(* CoDeSys 2.3.9.47 project: myhome.pro *)
(* Libraries: TcDatabase.lib 17.3.10 13:31:12, COMlibV2.lib 24.2.14 12:45:46, TcSUPS.lib 4.12.14 19:04:14, TcBaseMath.lib 27.7.04 12:07:56, TcMath.lib 23.9.04 15:15:30, TcBABasic.lib 29.5.12 16:01:34, TcBase.lib 14.5.09 12:14:08, TcSystem.lib 24.2.16 14:35:18, TcUtilities.lib 3.2.16 16:08:58, TcEL6851.lib 22.4.12 13:04:27, STANDARD.LIB 5.6.98 12:03:02, TcpIp.lib 9.1.14 13:33:22 *)

(* Global variable list: Global_Variables *)
VAR_GLOBAL

	SYS_VKE_0:		BOOL	:=	FALSE;		(*SYSTEM ALWAYS 0*)
	SYS_VKE_1:		BOOL	:=	TRUE;		(*SYSTEM ALWAYS 1*)
	SYS_IBN_1:		BOOL	:=	TRUE;		(*SYSTEM IBN ALWAYS 1*)

	di_System_Time:	DINT;

	SYS_FPE_100MS:	BOOL	:=	FALSE;		(*SYSTEM TIME 0.1 sec*)
	SYS_FPE_200MS:	BOOL	:=	FALSE;		(*SYSTEM TIME 0.2 sec*)
	SYS_FPE_500MS:	BOOL	:=	FALSE;		(*SYSTEM TIME 0.5 sec*)
	SYS_FPE_1S:		BOOL	:=	FALSE;		(*SYSTEM TIME 1.0 sec*)
	SYS_FPE_2S:		BOOL	:=	FALSE;		(*SYSTEM TIME 2.0 sec*)

	SYS_TOG_100MS:	BOOL	:=	FALSE;		(*SYSTEM TIME 0.1 sec*)
	SYS_TOG_200MS:	BOOL	:=	FALSE;		(*SYSTEM TIME 0.2 sec*)
	SYS_TOG_500MS:	BOOL	:=	FALSE;		(*SYSTEM TIME 0.5 sec*)
	SYS_TOG_1S:		BOOL	:=	FALSE;		(*SYSTEM TIME 1.0 sec*)
	SYS_TOG_2S:		BOOL	:=	FALSE;		(*SYSTEM TIME 2.0 sec*)

	SYS_T_100MS:		TON;					(*SYSTEM TIME 0.1 sec*)
	SYS_T_200MS:		TON;					(*SYSTEM TIME 0.2 sec*)
	SYS_T_500MS:		TON;					(*SYSTEM TIME 0.5 sec*)
	SYS_T_1S:			TON;					(*SYSTEM TIME 1.0 sec*)
	SYS_T_2S:			TON;					(*SYSTEM TIME 2.0 sec*)

	AX_FPE_100MS:	R_TRIG;				(*SYSTEM AUX FPE 0.1 sec*)
	AX_FPE_200MS:	R_TRIG;				(*SYSTEM AUX FPE 0.2 sec*)
	AX_FPE_500MS:	R_TRIG;				(*SYSTEM AUX FPE 0.5 sec*)
	AX_FPE_1S:		R_TRIG;				(*SYSTEM AUX FPE 1.0 sec*)
	AX_FPE_2S:		R_TRIG;				(*SYSTEM AUX FPE 2.0 sec*)

	bNightMode:	BOOL := FALSE;	(*limits Brightness if active*)
	fbTime : FB_LocalSystemTime := ( bEnable := TRUE, dwCycle := 1 );

(*DIGITAL INPUTS/Outputs*)
	(*SPS Switch 01 Arbeitsraum*)
	DI_S01_1 	AT %IX50.0 : BOOL;	(*Function Left 1*)
	DI_S01_2	AT %IX50.1 : BOOL;	(*Function Right 1*)
	DI_S01_3	AT %IX50.2 : BOOL;	(*Function Left 2*)
	DI_S01_4	AT %IX50.3 : BOOL;	(*Function Right 2*)
	DI_S01_5	AT %IX50.4 : BOOL;	(*Function Left 3*)
	DI_S01_6	AT %IX50.5 : BOOL;	(*Function Right 3*)
	DO_S01_0 	AT %QX50.0 : BOOL;	(*Status LED Left 1*)
	DO_S01_1 	AT %QX50.1 : BOOL;	(*Status LED Right 1*)
	DO_S01_2 	AT %QX50.2 : BOOL;	(*Status LED Left 2*)
	DO_S01_3 	AT %QX50.3 : BOOL;	(*Status LED Right 2*)
	DO_S01_4 	AT %QX50.4 : BOOL;	(*Status LED Left 3*)
	DO_S01_5 	AT %QX50.5 : BOOL;	(*Status LED Right 3*)
	DO_S01_6 	AT %QX50.6 : BOOL;	(*Background LED*)

	(*SPS Switch 02 Wohnzimmer*)
	DI_S02_1 	AT %IX50.6 : BOOL;	(*Function Left 1*)
	DI_S02_2	AT %IX50.7 : BOOL;	(*Function Right 1*)
	DI_S02_3	AT %IX51.0 : BOOL;	(*Function Left 2*)
	DI_S02_4	AT %IX51.1 : BOOL;	(*Function Right 2*)
	DI_S02_5	AT %IX51.2 : BOOL;	(*Function Left 3*)
	DI_S02_6	AT %IX51.3 : BOOL;	(*Function Right 3*)
	DO_S02_0 	AT %QX50.7 : BOOL;	(*Status LED Left 1*)
	DO_S02_1 	AT %QX51.0 : BOOL;	(*Status LED Right 1*)
	DO_S02_2 	AT %QX51.1 : BOOL;	(*Status LED Left 2*)
	DO_S02_3 	AT %QX51.2 : BOOL;	(*Status LED Right 2*)
	DO_S02_4 	AT %QX51.3 : BOOL;	(*Status LED Left 3*)
	DO_S02_5 	AT %QX51.4 : BOOL;	(*Status LED Right 3*)
	DO_S02_6 	AT %QX51.5 : BOOL;	(*Background LED*)

	(*DOUBLE Switch 03*)
	DI_S03_1 	AT %IX51.4 : BOOL;	(*Function Left*)
	DI_S03_2 	AT %IX51.5 : BOOL;	(*Function Right*)

	(*DOUBLE Switch 04*)
	DI_S04_1 	AT %IX51.6 : BOOL;	(*Function Left*)
	DI_S04_2 	AT %IX51.7 : BOOL;	(*Function Right*)

	(*SPS Switch 05 Schlafzimmer Bett Links*)
	DI_S05_1 	AT %IX52.0 : BOOL;	(*Function Left 1*)
	DI_S05_2	AT %IX52.1 : BOOL;	(*Function Right 1*)
	DI_S05_3	AT %IX52.2 : BOOL;	(*Function Left 2*)
	DI_S05_4	AT %IX52.3 : BOOL;	(*Function Right 2*)
	DI_S05_5	AT %IX52.4 : BOOL;	(*Function Left 3*)
	DI_S05_6	AT %IX52.5 : BOOL;	(*Function Right 3*)
	DO_S05_0 	AT %QX51.6 : BOOL;	(*Status LED Left 1*)
	DO_S05_1 	AT %QX51.7 : BOOL;	(*Status LED Right 1*)
	DO_S05_2 	AT %QX52.0 : BOOL;	(*Status LED Left 2*)
	DO_S05_3 	AT %QX52.1 : BOOL;	(*Status LED Right 2*)
	DO_S05_4 	AT %QX52.2 : BOOL;	(*Status LED Left 3*)
	DO_S05_5 	AT %QX52.3 : BOOL;	(*Status LED Right 3*)
	DO_S05_6 	AT %QX52.4 : BOOL;	(*Background LED*)

	(*SPS Switch 06 Schlafzimmer Bett Rechts*)
	DI_S06_1 	AT %IX52.6 : BOOL;	(*Function Left 1*)
	DI_S06_2	AT %IX52.7 : BOOL;	(*Function Right 1*)
	DI_S06_3	AT %IX53.0 : BOOL;	(*Function Left 2*)
	DI_S06_4	AT %IX53.1 : BOOL;	(*Function Right 2*)
	DI_S06_5	AT %IX53.2 : BOOL;	(*Function Left 3*)
	DI_S06_6	AT %IX53.3 : BOOL;	(*Function Right 3*)
	DO_S06_0 	AT %QX52.5 : BOOL;	(*Status LED Left 1*)
	DO_S06_1 	AT %QX52.6 : BOOL;	(*Status LED Right 1*)
	DO_S06_2 	AT %QX52.7 : BOOL;	(*Status LED Left 2*)
	DO_S06_3 	AT %QX53.0 : BOOL;	(*Status LED Right 2*)
	DO_S06_4 	AT %QX53.1 : BOOL;	(*Status LED Left 3*)
	DO_S06_5 	AT %QX53.2 : BOOL;	(*Status LED Right 3*)
	DO_S06_6 	AT %QX53.3 : BOOL;	(*Background LED*)

	(*DOUBLE Switch 07*)
	DI_S07_1 	AT %IX53.4 : BOOL;	(*Function Left*)
	DI_S07_2 	AT %IX53.5 : BOOL;	(*Function Right*)

	(*SINGLE Switch 08*)
	DI_S08	 	AT %IX53.6 : BOOL;	(*Function*)

	(*SINGLE Switch 09*)
	DI_S09	 	AT %IX53.7 : BOOL;	(*Function*)

	(*SINGLE Switch 10*)
	DI_S10	 	AT %IX54.0 : BOOL;	(*Function*)

	(*SINGLE Swith 11*)
	DI_S11	 	AT %IX54.1 : BOOL;	(*Function*)

	(*MOTION Swith 01*)
	DI_BM1	 	AT %IX54.3 : BOOL;	(*Function*)

	(*MOTION Swith 02*)
	DI_BM2	 	AT %IX54.4 : BOOL;	(*Function*)

	(*MOTION Swith 03*)
	DI_BM3	 	AT %IX54.5 : BOOL;	(*Function*)

	(*Relais*)
	DO_NN_K01	AT %QX54.0 : BOOL;	(*Relais Netzteil Arbeitsraum*)
	DO_NN_K02	AT %QX54.1 : BOOL;	(*Relais Steckdosen Arbeitsraum*)
	DO_NN_K03	AT %QX54.2 : BOOL;	(*Relais Netzteil Wohnzimmer*)
	DO_NN_K04	AT %QX54.3 : BOOL;	(*Relais Steckdosen Fernseher*)
	DO_NN_K05	AT %QX54.4 : BOOL;	(*Relais Netzteil Küche*)
	DO_NN_K06	AT %QX54.5 : BOOL;	(*Relais Netzteil Zimmer / Schlafzimmer*)
	DO_NN_K07	AT %QX54.6 : BOOL;	(*Relais Netzteil WC, Gang und Abstellraum*)
	DO_NN_K08	AT %QX54.7 : BOOL;	(*Relais Licht Bad*)
	DO_NN_K09	AT %QX53.6 : BOOL;	(*Relais Ventilator WC*)
	DO_NN_K10	AT %QX53.7 : BOOL;	(*Relais Reserve*)

	DO_NAS_BACKUP_ON_OFF	AT %QX53.4 : BOOL;	(*Relais NAS-Backup Pulse Power Switch*)
	DO_NAS_ON_OFF	AT %QX53.5 : BOOL;	(*Relais  NAS Pulse Power Switch*)

	fbPowerPC:PRG_FB_PULSE_SWITCH;
	fbPowerNAS:PRG_FB_PULSE_SWITCH;
	fbPowerNASBackup:PRG_FB_PULSE_SWITCH;

(* DMX Line *)
	fbEL6851Communication	:	FB_EL6851Communication;
	stDMXInDataLinie01               AT %I*	:	ST_EL6851InData;
	stDMXOutDataLinie01              AT %Q*	:	ST_EL6851OutData;
	stCommandBuffer01						:	ST_DMXCommandBuffer;
	arrDMXProcessData						:	ARRAY [1..512] OF BYTE;

(* 	I/O variables for a KL6001 terminal*)
	COMin_KL6001			AT %I* 	: KL6inData22B;		(* linked to the KL6001 in the TwinCAT System Manager *)
	COMout_KL6001		AT %Q*	: KL6outData22B;	(* linked to the KL6001 in the TwinCAT System Manager *)
	RxBuffer2: ComBuffer;	(* Receive data buffer; used with all receive function blocks *)
	TxBuffer2: ComBuffer;	(* Transmit data buffer; used with all receive function blocks *)

	COMin_COM4			AT %I* 	: KL6inData22B;		(* linked to the KL6001 in the TwinCAT System Manager *)
	COMout_COM4		AT %Q*	: KL6outData22B;	(* linked to the KL6001 in the TwinCAT System Manager *)

(*	FIFO for Trend if Database is off - Max 1 Week can be saved with 1 value every Minute*)
	TemperatureSchlafzimmerFIFO: PRG_FIFO_10080;
	TemperatureKinderzimmerFIFO: PRG_FIFO_10080;
	TemperatureKuecheFIFO: PRG_FIFO_10080;
	HumiditySchlafzimmerFIFO: PRG_FIFO_10080;
	HumidityKinderzimmerFIFO: PRG_FIFO_10080;
	HumidityKuecheFIFO: PRG_FIFO_10080;

	TemperatureTerrariumLinksFIFO: PRG_FIFO_10080;
	HumidityTerrariumLinksFIFO: PRG_FIFO_10080;
	TemperatureTerrariumRechtsFIFO: PRG_FIFO_10080;
	HumidityTerrariumRechtsFIFO: PRG_FIFO_10080;

(* TEST UDP*)
	g_sTcIpConnSvrAddr								:  T_AmsNetId := '10.0.0.6';

	(* Some project specific error codes *)
	PLCPRJ_ERROR_SENDFIFO_OVERFLOW		: UDINT := 16#8103;
	PLCPRJ_ERROR_RECFIFO_OVERFLOW		: UDINT := 16#8104;

END_VAR

VAR_GLOBAL CONSTANT
	bLogDebugMessages								: BOOL := TRUE;

	MAX_CLIENT_CONNECTIONS						: UDINT(1..20) := 5;
	MAX_PLCPRJ_RXBUFFER_SIZE					: UDINT := 1000;


	PLCPRJ_RECONNECT_TIME						: TIME := T#3s;
	PLCPRJ_SEND_CYCLE_TIME						: TIME := T#1s;
	PLCPRJ_ACCEPT_POLLING_TIME					: TIME := T#1s;

	PLCPRJ_RECEIVE_POLLING_TIME		 			: TIME := T#1s;
	PLCPRJ_RECEIVE_TIMEOUT						: TIME := T#50s;

	(* Some project specific error codes *)
	PLCPRJ_ERROR_RECEIVE_BUFFER_OVERFLOW	: UDINT := 16#8101; (* receive buffer overflow*)
	PLCPRJ_ERROR_RECEIVE_TIMEOUT				: UDINT := 16#8102;(* receive timeout error *)

END_VAR

(* Global variable list: TwinCAT_Configuration *)
(* Generated automatically by TwinCAT - (read only) *)
VAR_CONFIG
	.stDMXInDataLinie01 AT %IB56 : ST_EL6851InData;
	.stDMXOutDataLinie01 AT %QB56 : ST_EL6851OutData;
	.COMin_KL6001 AT %IB132 : KL6inData22B;
	.COMout_KL6001 AT %QB576 : KL6outData22B;
END_VAR

(* Data type *)
TYPE E_ClientServerSteps :
(
	UDP_STATE_IDLE		:= 0,
	UDP_STATE_CREATE_START,
	UDP_STATE_CREATE_WAIT,
	UDP_STATE_SEND_START,
	UDP_STATE_SEND_WAIT,
	UDP_STATE_RECEIVE_START,
	UDP_STATE_RECEIVE_WAIT,
	UDP_STATE_CLOSE_START,
	UDP_STATE_CLOSE_WAIT,
	UDP_STATE_ERROR
);
END_TYPE

(* Data type *)
TYPE E_ClientSteps :
(
	CLIENT_STATE_IDLE,
	CLIENT_STATE_CONNECT_START,
	CLIENT_STATE_CONNECT_WAIT,
	CLIENT_STATE_DATAEXCHA_START,
	CLIENT_STATE_DATAEXCHA_WAIT,
	CLIENT_STATE_CLOSE_START,
	CLIENT_STATE_CLOSE_WAIT,
	CLIENT_STATE_ERROR
);
END_TYPE

(* Data type *)
TYPE E_DataExchaSteps :
(
	DATAEXCHA_STATE_IDLE,
	DATAEXCHA_STATE_SEND_START,
	DATAEXCHA_STATE_SEND_WAIT,
	DATAEXCHA_STATE_RECEIVE_START,
	DATAEXCHA_STATE_RECEIVE_WAIT,
	DATAEXCHA_STATE_ERROR
);
END_TYPE

(* Data type *)
TYPE E_SampleState :(
        eIdle := 0,
        eWriteAppend := 1,
        eWriteUpdate := 2,
        eWriteRingBuffer := 3
);
END_TYPE

(* Data type *)
TYPE E_ServerSteps :
(
	SERVER_STATE_IDLE,
	SERVER_STATE_LISTENER_OPEN_START,
	SERVER_STATE_LISTENER_OPEN_WAIT,
	SERVER_STATE_REMOTE_CLIENTS_COMM,
	SERVER_STATE_REMOTE_CLIENTS_CLOSE,
	SERVER_STATE_LISTENER_CLOSE_START,
	SERVER_STATE_LISTENER_CLOSE_WAIT,
	SERVER_STATE_ERROR
);
END_TYPE

(* Data type *)
TYPE E_SQLStatement :(
        eSQL_INSERT := 0,
        eSQL_SELECT := 1
);
END_TYPE

(* Data type *)
TYPE ST_FifoEntry :
STRUCT
	sRemoteHost		: STRING(15);		(* Remote address. String containing an (Ipv4) Internet Protocol dotted address. *)
	nRemotePort		: UDINT;			(* Remote Internet Protocol (IP) port. *)
	msg				: STRING;			(* Udp packet data *)
END_STRUCT
END_TYPE

(* Data type *)
TYPE ST_Record :
STRUCT
        Timestamp : DT;
        PLC_Value1 : REAL;
        PLC_Value2 : REAL;
        PLC_Value3 : REAL;
        PLC_Value4 : STRING;
END_STRUCT
END_TYPE

(* Data type *)
TYPE T_TimeStampLength : STRING(19);
END_TYPE

(* Data type *)
TYPE Type_HSV :
STRUCT
	Hue	:			REAL;
	Saturation:		REAL:= 100.0;
	Brightness:		REAL:=100.0;
END_STRUCT
END_TYPE

(* Data type *)
TYPE Type_LED :
STRUCT
	Switch_ON:			BOOL;
	Switch_RANDOM:		BOOL;
	bLight:				BOOL;
	Config:				Type_LED_CONFIG;
	Value:				REAL:=100;
	Brightness:			BYTE;
	fbDimmer2Switch: FB_Dimmer2Switch;
	fpSwitchOnOff: F_TRIG;
END_STRUCT
END_TYPE

(* Data type *)
TYPE Type_LED_CONFIG :
STRUCT
	tDimmTime: 		REAL	:= 5000;
	bDimmOnMode:	BOOL	:= TRUE;
	tDimmOnTime:		REAL	:= 500;
	bDimmOffMode:	BOOL	:= TRUE;
	tDimmOffTime:		REAL	:= 1000;
	Brightness_MAX	:REAL:=255;
END_STRUCT
END_TYPE

(* Data type *)
TYPE Type_LED_RGB :
STRUCT
	Hue				:REAL;
	Saturation			:REAL:= 100.0;
	Brightness			:REAL:=100;
	Switch_ON			:BOOL;
	Switch_RANDOM	:BOOL;
	bLight:			BOOL;
	Config				:Type_LED_RGB_CONFIG;
	Red					:BYTE;
	Green				:BYTE;
	Blue					:BYTE;
END_STRUCT
END_TYPE

(* Data type *)
TYPE Type_LED_RGB_CONFIG :
STRUCT
	Speed_RANDOM	:REAL;

	tDimmTime: 		REAL	:= 5000;
	bDimmOnMode:	BOOL	:= TRUE;
	tDimmOnTime:		REAL	:= 500;
	bDimmOffMode:	BOOL	:= TRUE;
	tDimmOffTime:		REAL	:= 1000;
END_STRUCT
END_TYPE

(* Data type *)
TYPE Type_LED_RGB_with_FB :
STRUCT
	Hue				:REAL;
	Saturation			:REAL:= 100.0;
	Brightness			:REAL:=100;
	Switch_ON			:BOOL;
	Switch_RANDOM	:BOOL;
	bLight:			BOOL;
	Config				:Type_LED_RGB_CONFIG;
	Red					:BYTE;
	Green				:BYTE;
	Blue					:BYTE;
	fbDimmer2Switch: FB_Dimmer2Switch;
	fpSwitchOnOff: F_TRIG;
END_STRUCT
END_TYPE

(* Data type *)
TYPE Type_SCENE_CONFIG :
STRUCT
	tDimmTime: 		REAL	:= 5000;
	bDimmOnMode:	BOOL	:= TRUE;
	tDimmOnTime:		REAL	:= 500;
	bDimmOffMode:	BOOL	:= TRUE;
	tDimmOffTime:		REAL	:= 1000;
END_STRUCT
END_TYPE

(* Data type *)
TYPE Type_SCENE_WZ :
STRUCT
	tyMirror1 : Type_LED_RGB;
	tyMirror2 : Type_LED_RGB;
	tyMirror3 : Type_LED_RGB;
(*tyCeiling : Type_LED_RGB;*)
END_STRUCT
END_TYPE

(* POU MAIN, ST *)
PROGRAM MAIN
VAR
	nCount 						: UDINT;
	tGlobOff:	TON;
	tGlobOffLong:	TOF;
	fnGlobOff: R_TRIG;

	nBrightness1:BYTE;
	nBrightness2:BYTE;
	nBrightness3:BYTE;
	nBrightness4:BYTE;
	nBrightness5:BYTE;
	nBrightness6:BYTE;
	nBrightness7:BYTE;
	nBrightness8:BYTE;
	nBrightness9:BYTE;

	READ_TEMP_HUM:SYS_03_READ_TEMP_HUM;
	COMM_XMC : SYS_02_COMM_XMC;

END_VAR
SYS_00_BASICS();
READ_TEMP_HUM(bEnable:=TRUE );
COMM_XMC(bEnable:=TRUE );

tGlobOff(IN:= DI_S05_6 OR DI_S06_6, PT:= T#2s);
fnGlobOff(CLK:= tGlobOff.Q );
tGlobOffLong(IN:= fnGlobOff.Q, PT:= T#4s);

(*Aufruf Wohnräume*)
ROOM_01_ARBEITSZIMMER(ibGlobOff:= fnGlobOff.Q, ibGlobOffLong:= tGlobOffLong.Q);
ROOM_02_WOHNZIMMER(ibGlobOff:= fnGlobOff.Q, ibGlobOffLong:= tGlobOffLong.Q, irTemperature:=READ_TEMP_HUM.Temp[1], irHumidity:=READ_TEMP_HUM.Humidity[1]);
ROOM_03_KUECHE(ibGlobOff:= fnGlobOff.Q, ibGlobOffLong:= tGlobOffLong.Q, irTemperature:=READ_TEMP_HUM.Temp[4], irHumidity:=READ_TEMP_HUM.Humidity[4]);
ROOM_04_ZIMMER(ibGlobOff:= fnGlobOff.Q, ibGlobOffLong:= tGlobOffLong.Q, irTemperature:=READ_TEMP_HUM.Temp[1], irHumidity:=READ_TEMP_HUM.Humidity[1], irTemperatureSZ:=READ_TEMP_HUM.Temp[5], irHumiditySZ:=READ_TEMP_HUM.Humidity[5]);
ROOM_05_WC_GANG(ibGlobOff:= fnGlobOff.Q, ibGlobOffLong:= tGlobOffLong.Q);

DO_S05_5:=	(ROOM_01_ARBEITSZIMMER.obDevOn OR ROOM_02_WOHNZIMMER.obDevOn OR
			ROOM_03_KUECHE.obDevOn OR ROOM_04_ZIMMER.obDevOn OR
			ROOM_05_WC_GANG.obDevOn) AND (fbTime.systemTime.wHour < 6 OR fbTime.systemTime.wHour >= 22);

DO_S06_5:=	(ROOM_01_ARBEITSZIMMER.obDevOn OR ROOM_02_WOHNZIMMER.obDevOn OR
			ROOM_03_KUECHE.obDevOn OR ROOM_04_ZIMMER.obDevOn OR
			ROOM_05_WC_GANG.obDevOn) AND (fbTime.systemTime.wHour < 6 OR fbTime.systemTime.wHour >= 22);

arrDMXProcessData[128] := nBrightness1;
arrDMXProcessData[129] := nBrightness2;
arrDMXProcessData[130] := nBrightness3;
arrDMXProcessData[131] := nBrightness4;
arrDMXProcessData[132] := nBrightness5;
arrDMXProcessData[133] := nBrightness6;
arrDMXProcessData[134] := nBrightness7;
arrDMXProcessData[135] := nBrightness8;

fbEL6851Communication(	wSourceManufacturerID := 16#42_41,
						dwSourceDeviceID := 16#12_13_14_15,
						bEnableSendingData := TRUE,
						bSetCycleMode := TRUE,
						bSendDefaultData := FALSE,
						uiDataLength := 512,
						dwOptions := 0,
						stEL6851InData := stDMXInDataLinie01,
						stEL6851OutData := stDMXOutDataLinie01,
						stCommandBuffer := stCommandBuffer01,
						arrProcessData := arrDMXProcessData);

fbTime();

SYS_01_TREND(
	irTemperatureSchlafzimmer:= READ_TEMP_HUM.Temp[5],
	irHumiditySchlafzimmer:= READ_TEMP_HUM.Humidity[5],
	irTemperatureKinderzimmer:= READ_TEMP_HUM.Temp[1],
	irHumidityKinderzimmer:= READ_TEMP_HUM.Humidity[1],
	irTemperatureKueche:= READ_TEMP_HUM.Temp[4],
	irHumidityKueche:= READ_TEMP_HUM.Humidity[4],
	irTemperatureTerrariumLinks:=COMM_XMC.TemperatureTerrariumLinks,
	irHumidityTerrariumLinks:=COMM_XMC.HumidityTerrariumLinks,
	irTemperatureTerrariumRechts:=COMM_XMC.TemperatureTerrariumRechts,
	irHumidityTerrariumRechts:=COMM_XMC.HumidityTerrariumRechts);
END_PROGRAM

(* POU General/SYS_03_READ_TEMP_HUM, ST *)
FUNCTION_BLOCK SYS_03_READ_TEMP_HUM
VAR_INPUT
	bEnable:BOOL;
END_VAR
VAR_OUTPUT
END_VAR
VAR
	Timer: TON;
	iActSensorNumber:UINT:=1;
	iNumberOfSensors:UINT:=5;
	RequestString:STRING;
	Send: SendString;
	SendBusy: BOOL;
	SendErrorID: ComError_t;

	Receive: ReceiveString;
	ReceivedString: STRING;
	LastReceivedString: STRING;
	StringReceived: BOOL;
	ReceiveBusy: BOOL;
	ReceiveError: BOOL;
	ReceiveErrorID: ComError_t;
	ReceiveTimeout: BOOL;
	ReceiveCounter: UDINT;
END_VAR
VAR PERSISTENT
	TempOffset: ARRAY [1..10] OF REAL := 0;
	Temp: ARRAY [1..10] OF REAL := 0;
	RecTempStr: ARRAY [1..10] OF STRING;
	Humidity: ARRAY [1..10] OF REAL := 0;
	RecHumidityStr: ARRAY [1..10] OF STRING;
END_VAR
(*==================================================================
	Call the send block every second to repeat the transmission.
	Also call the block as long as it is busy to finish a transmission.
*)

TempOffset[1]:=-1.2;
TempOffset[2]:=-2.6;
TempOffset[3]:=-1.6;
TempOffset[4]:=-2.6;
TempOffset[5]:=-1;

Timer(IN:=bEnable, PT:=T#1s);

IF Timer.Q OR Send.Busy THEN

	iActSensorNumber:=iActSensorNumber+1;
	IF iActSensorNumber > iNumberOfSensors THEN
		iActSensorNumber:=1;
	END_IF

	RequestString:= CONCAT('s',UINT_TO_STRING(iActSensorNumber));

	Send(	SendString:= RequestString,
			TXbuffer:= TxBuffer2,	(* see global variables *)
			Busy=> SendBusy,
			Error=> SendErrorID);

	Timer(IN:=FALSE); (* reset timer *)
END_IF

(*==================================================================
	Receive string data 
	The block receives any data strings beginning with a STX ($02) character and 
	ending with an ETX ($03) character.	
*)
Receive(
	Prefix:= '$02',
	Suffix:= '$03',
	Timeout:= T#1s,
	ReceivedString:= ReceivedString,
	RXbuffer:= RxBuffer2,
	StringReceived=> StringReceived,
	Busy=> ReceiveBusy,
	Error=> ReceiveErrorID,
	RxTimeout=> ReceiveTimeout );
IF StringReceived THEN
	ReceiveCounter := ReceiveCounter + 1;
	LastReceivedString := ReceivedString;

	(*Extract Temperatur Value from received String*)
	(*Nr. 4 = Küche, Nr.5 = Schlafzimmer*)
	RecTempStr[iActSensorNumber] := MID (ReceivedString,4,5);
	Temp[iActSensorNumber]:=STRING_TO_REAL(RecTempStr[iActSensorNumber] )+TempOffset[iActSensorNumber];

	(*Extract Humidity Value from received String*)
	RecHumidityStr[iActSensorNumber] := MID (ReceivedString,4,16);
	Humidity[iActSensorNumber]:=STRING_TO_REAL(RecHumidityStr[iActSensorNumber] );
END_IF


(*==================================================================
	Background communication with the KL6001 terminal.
	Please check the FAST program where the background communication with the
	KL6001 terminal is processed in a separate fast task. A fast task is in this case 
	necessary to guarantee an acceptable transfer rate.
*)
END_FUNCTION_BLOCK

(* POU General/SYS_02_COMM_XMC, ST *)
FUNCTION_BLOCK SYS_02_COMM_XMC
VAR_INPUT
	bEnable:BOOL;
END_VAR
VAR_OUTPUT
END_VAR
VAR
	Timer: TON;
	fpSend: R_TRIG;
	fpSwitchRollo: R_TRIG;
	fpAutoUp: R_TRIG;
	CommandString:STRING;
	Send: SendString;
	SendBusy: BOOL;
	SendErrorID: ComError_t;

	Receive: ReceiveString;
	ReceivedString: STRING;
	LastReceivedString: STRING;
	StringReceived: BOOL;
	ReceiveBusy: BOOL;
	ReceiveError: BOOL;
	ReceiveErrorID: ComError_t;
	ReceiveTimeout: BOOL;
	ReceiveCounter: UDINT;

	(* communication buffer between application and SerialLineControl *)
	RxBuffer		:ComBuffer;
	TxBuffer		:ComBuffer;

	(* serial line control *)
	fbLineCtrlAds	:SerialLineControlADS;
	bAdsError		:BOOL;
	nAdsErrorID		:UDINT;
	sNetId			:T_AmsNetId;
	stSerialCfg		:ComSerialConfig;

	bSendCommand:BOOL;

	boolRolloUp: BOOL := TRUE;
	boolRolloDown: BOOL;
	boolRolloCoUp: BOOL;
	boolRolloCoDown: BOOL;
	TON_DriveTime : TON;

	nRolloStat:INT:=10;
	nFindString : INT;


	TemperatureTerrariumLinks: REAL;
	HumidityTerrariumLinks: REAL;
	TemperatureTerrariumRechts: REAL;
	HumidityTerrariumRechts: REAL;
	tmpString: STRING;
	tmpString1: STRING;
END_VAR
VAR CONSTANT
	bRolloAutoControl:BOOL;
	nRolloAutoOpenTime:INT;
	ROLLO_UP : INT :=10;
	ROLLO_DRIVE_UP : INT := 11;
	ROLLO_DOWN : INT := 20;
	ROLLO_DRIVE_DOWN: INT := 21;
END_VAR
stSerialCfg.ComPort := 4;

fbLineCtrlAds(
	Connect:= bEnable,
	SerialCfg:= stSerialCfg,
	NetId:= sNetId,
	Timeout:= ,
	TxBuffer:= TxBuffer,
	RxBuffer:= RxBuffer,
	PortOpened=> ,
	Error=> bAdsError,
	ErrorID=> nAdsErrorID,
	Busy=> ,
	TxBufCount=> ,
	RxBufCount=> );

(*==================================================================
	Senden der Befehle	
	Befehle: CO_U: Rollo hoch, CU_D: Rollo runter, CO_S: Rollo Stop
*)
fpSend(CLK:=bSendCommand);
IF fpSend.Q OR Send.Busy OR Timer.Q THEN
	Send(	SendString:= CommandString,
			TXbuffer:= TxBuffer,	(* see global variables *)
	Busy=> SendBusy,
	Error=> SendErrorID);

	Timer(IN:=FALSE, PT:=T#10s);
END_IF

(*==================================================================
	Steuerung der Rollo
	Rauf-, Runterfahren und Stop	
*)

(*Schalter Rollo*)
fpSwitchRollo(CLK:= DI_S02_6);
Timer(IN:=bSendCommand, PT:=T#10s);

IF StringReceived THEN
	ReceiveCounter := ReceiveCounter + 1;
	LastReceivedString := ReceivedString;
END_IF

(*Um 10 Uhr automatisch die Rollo öffnen*)
fpAutoUp(CLK:= (fbTime.systemTime.wHour = nRolloAutoOpenTime) AND bRolloAutoControl);
IF fpAutoUp.Q THEN
	nRolloStat := ROLLO_DOWN;
END_IF


CASE nRolloStat OF
	ROLLO_UP:
		(*Rollo ist oben, starte Runterfahren bei Knopfdruck*)
		IF fpSwitchRollo.Q THEN
			CommandString:= 'CO_D';
			bSendCommand := TRUE;
		END_IF

		(*Befehl ist gesendet, warte auf Rückmeldung*)
		IF StringReceived THEN
			nFindString := FIND(LastReceivedString, 'CO_D');
			IF nFindString > 0 THEN
				nRolloStat := ROLLO_DRIVE_DOWN;
			END_IF
			bSendCommand := FALSE;
		END_IF

	ROLLO_DRIVE_DOWN:
		(*Starte Zeit*)
		IF NOT bSendCommand THEN
			TON_DriveTime(IN:= TRUE, PT:=T#21s);
		END_IF
		DO_S02_5 := SYS_TOG_200MS;

		(*Wenn während dem Fahren der Knopf gedrückt wird, dann wird Stop gesendet.*)
		IF fpSwitchRollo.Q THEN
			CommandString:= 'CO_S';
			bSendCommand := TRUE;
		END_IF

		(*Zeit abgelaufen, Rollo ist oben*)
		IF TON_DriveTime.Q THEN
			TON_DriveTime(IN:= FALSE);
			nRolloStat := ROLLO_DOWN;
			DO_S02_5:=FALSE;
		END_IF

		(*Wenn Stop Befehl gesendet wurde, dann springe zu status ROLLO_UP, dass beim nächsten druck das Rollo weiter nach unten fährt*)
		IF StringReceived THEN
			nFindString := FIND(LastReceivedString, 'CO_S');
			IF nFindString > 0 THEN
				nRolloStat := ROLLO_UP;
				DO_S02_5:=FALSE;
			END_IF
			bSendCommand := FALSE;
		END_IF

	ROLLO_DOWN:
		(*Rollo ist unten, starte Raufahren bei Knopfdruck*)
		IF fpSwitchRollo.Q OR  fpAutoUp.Q THEN
			CommandString:= 'CO_U';
			bSendCommand := TRUE;
		END_IF

		(*Befehl ist gesendet, warte auf Rückmeldung*)
		IF StringReceived THEN
			nFindString := FIND(LastReceivedString, 'CO_U');
			IF nFindString > 0 THEN
				nRolloStat := ROLLO_DRIVE_UP;
			END_IF
			bSendCommand := FALSE;
		END_IF

	ROLLO_DRIVE_UP:
		(*Starte Zeit*)
		IF NOT bSendCommand THEN
			TON_DriveTime(IN:= TRUE, PT:=T#23s);
		END_IF
		DO_S02_5 := SYS_TOG_100MS;

		(*Wenn während dem Fahren der Knopf gedrückt wird, dann wird Stop gesendet.*)
		IF fpSwitchRollo.Q THEN
			CommandString:= 'CO_S';
			bSendCommand := TRUE;
		END_IF

		(*Zeit abgelaufen, Rollo ist oben*)
		IF TON_DriveTime.Q THEN
			TON_DriveTime(IN:= FALSE);
			nRolloStat := ROLLO_UP;
			DO_S02_5:=FALSE;
		END_IF

		(*Wenn Stop Befehl gesendet wurde, dann springe zu status ROLLO_DOWN, dass beim nächsten druck das Rollo weiter nach oben fährt*)
		IF StringReceived THEN
			nFindString := FIND(LastReceivedString, 'CO_S');
			IF nFindString > 0 THEN
				nRolloStat := ROLLO_DOWN;
				DO_S02_5:=FALSE;
			END_IF
			bSendCommand := FALSE;
		END_IF
END_CASE

IF bSendCommand THEN
	DO_S02_5 := TRUE;
END_IF


(*Daten vom Terrarium extrahieren*)
nFindString := FIND(LastReceivedString, 'Terrarium');
IF nFindString > 0 THEN
	tmpString := DELETE(LastReceivedString, 11,1);
	TemperatureTerrariumRechts := STRING_TO_REAL(MID(tmpString,FIND(tmpString, ' '),1));
	tmpString := DELETE(tmpString, FIND(tmpString, ' '),1);
	HumidityTerrariumRechts := STRING_TO_REAL(MID(tmpString,FIND(tmpString1, ' '),1));
	tmpString := DELETE(tmpString, FIND(tmpString, ' '),1);
	TemperatureTerrariumLinks := STRING_TO_REAL(MID(tmpString,FIND(tmpString1, ' '),1));
	tmpString := DELETE(tmpString, FIND(tmpString, ' '),1);
	HumidityTerrariumLinks := STRING_TO_REAL(MID(tmpString,FIND(tmpString1, ' '),1));
	LastReceivedString := '';
END_IF


(*==================================================================
	Receive string data 
	The block receives any data strings beginning with a STX ($02) character and 
	ending with an ETX ($03) character.	
*)

Receive(
	Prefix:= '$02',
	Suffix:= '$03',
	Timeout:= T#1s,
	ReceivedString:= ReceivedString,
	RXbuffer:= RxBuffer,
	StringReceived=> StringReceived,
	Busy=> ReceiveBusy,
	Error=> ReceiveErrorID,
	RxTimeout=> ReceiveTimeout );
END_FUNCTION_BLOCK

(* POU General/SYS_00_BASICS, ST *)
PROGRAM SYS_00_BASICS
VAR
	T_100ms_TON: TON;
	T_100ms_TOF: TOF;

(* UPS related ... *)
	fbUPS			: FB_S_UPS;			(* UPS-FB instance *)
					(* Default Values of FB_S_UPS-Inputs:
						sNetID 			:= '' ==> local netid
						iPLCPort 		:= AMSPORT_R0_PLC_RTS1 ==> 801 = 1st Runtime System
						iUPSPort		:= 16#4A8 ==> Port for reading Power State of UPS
						tTimeout 		:= DEFAULT_ADS_TIMEOUT ==> 5S
						eUpsMode 		:= eSUPS_WrPersistData_Shutdown ==> writing persistent data + shutdown
						ePersistentMode := SPDM_2PASS ==> All data is from same plc cycle, cycletime exceeds possible. Plc stops with the shutdown, a few cycles after writing persistent data. 
						tRecoverTime 	:= T#10s ==> 10s power to recover from short power failure before eSUPS_PowerOK is reported (in mode eSUPS_WrPersistData_NoShutdown/eSUPS_CheckPowerStatus)
					*)
	eUpsMode		: E_S_UPS_Mode	:= eSUPS_WrPersistData_Shutdown; (* UPS mode (writing persistent data + shutdown) *)

	(* !!! TO DO: REPLACE WITH YOUR PLC VARIABLES/FB INSTANCES !!! regular PLC variables/FB instances ... *)
	iCounter		: UDINT;					(* non persistent counter *)

END_VAR

VAR PERSISTENT
	(* !!! TO DO: REPLACE WITH YOUR PERSISTENT PLC VARIABLES !!! persistent variables ... *)
	iPowerFailureCount: UDINT:=0; (* persistent counter of power failures *)
END_VAR
SYS_VKE_0		:=	FALSE;
SYS_VKE_1		:=	TRUE;
SYS_IBN_1		:=	TRUE;

di_System_Time := TIME_TO_DINT(TIME());


(*GENERATE SYSTEM PULSE FLAGS*)

SYS_T_100MS(IN:= SYS_IBN_1 AND NOT SYS_T_100MS.Q, PT:= T#100MS);
SYS_T_200MS(IN:= SYS_IBN_1 AND NOT SYS_T_200MS.Q, PT:= T#200MS);
SYS_T_500MS(IN:= SYS_IBN_1 AND NOT SYS_T_500MS.Q, PT:= T#500MS);
SYS_T_1S(IN:= SYS_IBN_1 AND NOT SYS_T_1S.Q, PT:= T#1S);
SYS_T_2S(IN:= SYS_IBN_1 AND NOT SYS_T_2S.Q, PT:= T#2S);

IF SYS_T_100MS.Q	THEN
	IF SYS_TOG_100MS THEN
		SYS_TOG_100MS := FALSE; 	ELSE	SYS_TOG_100MS := TRUE;
	END_IF
END_IF

IF SYS_T_200MS.Q	THEN
	IF SYS_TOG_200MS THEN
		SYS_TOG_200MS := FALSE; 	ELSE	SYS_TOG_200MS := TRUE;
	END_IF
END_IF

IF SYS_T_500MS.Q	THEN
	IF SYS_TOG_500MS THEN
		SYS_TOG_500MS := FALSE; 	ELSE	SYS_TOG_500MS := TRUE;
	END_IF
END_IF

IF SYS_T_1S.Q	THEN
	IF SYS_TOG_1S THEN
		SYS_TOG_1S := FALSE; 	ELSE	SYS_TOG_1S := TRUE;
	END_IF
END_IF

IF SYS_T_2S.Q	THEN
	IF SYS_TOG_2S THEN
		SYS_TOG_2S := FALSE; 	ELSE	SYS_TOG_2S := TRUE;
	END_IF
END_IF

AX_FPE_100MS(CLK:= SYS_TOG_100MS , Q=> SYS_FPE_100MS);
AX_FPE_200MS(CLK:= SYS_TOG_200MS , Q=> SYS_FPE_200MS);
AX_FPE_500MS(CLK:= SYS_TOG_500MS , Q=> SYS_FPE_500MS);
AX_FPE_1S(CLK:= SYS_TOG_1S , Q=> SYS_FPE_1S);
AX_FPE_2S(CLK:= SYS_TOG_2S , Q=> SYS_FPE_2S);

(* S-UPS Demo *)

(* call UPS-FB instance in first lines of the fastest PLC Task *)
fbUPS(eUpsMode := eUpsMode);
(* eUpsMode =							in case of powerfailure:
	 eSUPS_WrPersistData_Shutdown 		 	writing of persistent data + shutdown
	 eSUPS_WrPersistData_NoShutdown 		writing of PERSISTENT data, no shutdown
	 eSUPS_CheckPowerStatus 				reports powerfailure without ACTION (no writing, no shutdown) 
	 eSUPS_ImmediateShutdown 				skips writing of data, immediate shutdown
*)

(* evaluate UPS State *)
IF eGlobalSUpsState = eSUPS_PowerFailure THEN
	(* first cycle of powerfailure *)

	(* execute code that should only be done once with each powerfailure, i.e. increase powerfailure counter *)
	iPowerFailureCount := iPowerFailureCount + 1;
END_IF
END_PROGRAM

(* POU Rooms/ROOM_01_ARBEITSZIMMER, ST *)
PROGRAM ROOM_01_ARBEITSZIMMER
VAR_INPUT
	ibGlobOff:		BOOL;
	ibGlobOffLong:	BOOL;
END_VAR
VAR PERSISTENT
	fbWhiteCeiling: PRG_FB_LED_SINGLE;
	fbWhiteWorkplace: PRG_FB_LED_SINGLE;
	fbWhiteRegal: PRG_FB_LED_SINGLE;
	fbWhiteAbstellraum: PRG_FB_LED_SINGLE;


END_VAR
VAR
	fpBM1:R_TRIG;
	fnBM1:F_TRIG;
	tDoffBM1: TOF;
	boolAbstellraumEin: BOOL;
END_VAR
VAR_OUTPUT
	obDevOn:	BOOL;
END_VAR
(*LED light white ceiling*)
fbWhiteCeiling(
	i_bSwitchOn:= FALSE,
	i_bSwitchOff:= ibGlobOff,
	i_bSwitchOnOff:=  DI_S01_1,
	i_iSceneValue:= );

DO_S01_0 := fbWhiteCeiling.bLight;

(*LED light white workplace*)
fbWhiteWorkplace(
	i_bSwitchOn:= FALSE,
	i_bSwitchOff:= ibGlobOff,
	i_bSwitchOnOff:= DI_S01_2,
	i_iSceneValue:= );

DO_S01_1 := fbWhiteWorkplace.bLight;

(*LED light white Regal*)
fbWhiteRegal(
	i_bSwitchOn:= FALSE,
	i_bSwitchOff:= ibGlobOff,
	i_bSwitchOnOff:=DI_S02_2,
	i_iSceneValue:= );

DO_S02_1 := fbWhiteRegal.bLight;

(*flags of BM*)
tDoffBM1(IN:= DI_BM1, PT:= T#1s);

fpBM1(CLK:= tDoffBM1.Q);
fnBM1(CLK:= tDoffBM1.Q);

(*LED light white Abstellraum*)
fbWhiteAbstellraum(
	i_bSwitchOn:=fpBM1.Q AND NOT boolAbstellraumEin,
	i_bSwitchOff:=(fnBM1.Q AND NOT boolAbstellraumEin) OR ibGlobOff,
	i_bSwitchOnOff:=boolAbstellraumEin,
	i_iSceneValue:= );

(*relay for power supply*)
DO_NN_K01 :=	fbWhiteCeiling.bLight OR fbWhiteWorkplace.bLight OR fbWhiteRegal.bLight OR
				fbWhiteAbstellraum.bLight;

(*relay for power supply PC*)
fbPowerPC(bTrigPlug:= (DI_S01_6  OR (fbPowerPC.bStat AND DI_S05_5)) , bSwitchAck:= , bRelay=> DO_NN_K02);
DO_S01_5 := fbPowerPC.bStat;
DO_S05_4 := fbPowerPC.bStat  AND (fbTime.systemTime.wHour < 6 OR fbTime.systemTime.wHour >= 22);;


(*POWER NAS*)
fbPowerNAS(bTrigPlug:= DI_S01_4 OR (fbPowerNAS.bStat AND ibGlobOffLong), bSwitchAck:= , bRelay=> DO_NAS_ON_OFF, bStat=> DO_S01_3);
fbPowerNASBackup(bTrigPlug:= DI_S01_5 OR (fbPowerNASBackup.bStat AND ibGlobOffLong), bSwitchAck:= , bRelay=> DO_NAS_BACKUP_ON_OFF, bStat=> DO_S01_4);

(*DMX communication*)
arrDMXProcessData[1] := fbWhiteCeiling.Brightness;
arrDMXProcessData[2] := fbWhiteWorkplace.Brightness;
arrDMXProcessData[3] := fbWhiteAbstellraum.Brightness;
arrDMXProcessData[4] := fbWhiteRegal.Brightness;
arrDMXProcessData[200] := fbWhiteRegal.Brightness;

obDevOn:=		fbWhiteCeiling.bLight OR fbWhiteWorkplace.bLight OR fbWhiteRegal.bLight OR
				fbWhiteAbstellraum.bLight OR fbPowerPC.bStat OR fbPowerNAS.bStat;
END_PROGRAM

(* POU Own PRG's and FB's/PRG_FB_LED_SINGLE, ST *)
FUNCTION_BLOCK PRG_FB_LED_SINGLE
VAR_INPUT
	i_bSwitchOn:		BOOL;
	i_bSwitchOff:		BOOL;
	i_bSwitchOnOff:	BOOL;
	i_iSceneValue:	INT;
END_VAR
VAR_OUTPUT
END_VAR
VAR
	Switch_ON:			BOOL;
	Switch_RANDOM:		BOOL;
	bLight:				BOOL;
	bDimmUp:			BOOL;
	bDimmDown:			BOOL;
	nDimmStep:			INT := 10;
	Config:				Type_LED_CONFIG;
	Value:				REAL:=100;
	Brightness:			BYTE;
	fbDimmer2Switch: FB_Dimmer2Switch;
	fnSwitchOnOff: F_TRIG;
	fpSwitchOnOff: R_TRIG;
	fnSwitchOn: F_TRIG;
	fnSwitchOff: F_TRIG;
	tiLongSwitchOnOff:	TON;
	tiLongSwitchOn:	TON;
	tiLongSwitchOff:	TON;
END_VAR
(*dimm up and down*)
bDimmUp := (tiLongSwitchOn.Q OR (tiLongSwitchOnOff.Q AND nDimmStep = 10)) AND NOT bDimmDown;
bDimmDown := (tiLongSwitchOff.Q OR (tiLongSwitchOnOff.Q AND nDimmStep = 20)) AND NOT bDimmUp;

(*flag negative edge and timer of switch for on*)
tiLongSwitchOn(IN:= i_bSwitchOn, PT:= T#500ms);
fnSwitchOn(CLK:= i_bSwitchOn );

(*flag negative edge and timer of switch for off*)
tiLongSwitchOff(IN:= i_bSwitchOff, PT:= T#500ms);
fnSwitchOff(CLK:= i_bSwitchOff );

(*flag negative edge and timer of switch for on and off*)
tiLongSwitchOnOff(IN:= i_bSwitchOnOff, PT:= T#500ms);
fnSwitchOnOff(CLK:= i_bSwitchOnOff );

(*nDimmStep = 20 ----> dimm down*)
IF tiLongSwitchOnOff.Q AND fbDimmer2Switch.nOut = 100  AND fpSwitchOnOff.Q THEN
	nDimmStep := 20;
END_IF

(*nDimmStep = 10 ----> dimm up*)
fpSwitchOnOff(CLK:= tiLongSwitchOnOff.Q );
IF tiLongSwitchOnOff.Q AND fbDimmer2Switch.nOut = 0 AND fpSwitchOnOff.Q THEN
	nDimmStep := 10;
END_IF

(*switch light on*)
IF fnSwitchOn.Q OR ( fnSwitchOnOff.Q AND NOT  bLight) THEN
	 Switch_ON := TRUE;
END_IF

(*switch light off*)
IF (fnSwitchOff.Q AND NOT bDimmDown) OR ((fnSwitchOnOff.Q  AND NOT bDimmDown AND NOT bDimmUp) AND bLight) THEN
	 Switch_ON := FALSE;
END_IF

 fbDimmer2Switch(
	bSwitchDimmUp:= bDimmUp,
	bSwitchDimmDown:= bDimmDown,
	bOn:=  Switch_ON,
	bOff:= NOT  Switch_ON,
	bSetDimmValue:= FALSE,
	nDimmValue:= 0,
	tSwitchOverTime:=T#300MS ,
	tDimmTime:= REAL_TO_TIME( Config.tDimmTime),
	bMemoryModeOn:= TRUE,
	nOnValueWithoutMemoryMode:= 0,
	bDimmOnMode:=  Config.bDimmOnMode,
	tDimmOnTime:= REAL_TO_TIME( Config.tDimmOnTime),
	bDimmOffMode:=  Config.bDimmOffMode,
	tDimmOffTime:= REAL_TO_TIME( Config.tDimmOffTime),
	nOutMin:= 0,
	nOutMax:=REAL_TO_UINT(Value),
	bLight=>  bLight);

 Brightness := REAL_TO_BYTE(UINT_TO_REAL( fbDimmer2Switch.nOut)/100* Config.Brightness_MAX);
END_FUNCTION_BLOCK

(* POU Rooms/ROOM_02_WOHNZIMMER, ST *)
PROGRAM ROOM_02_WOHNZIMMER
VAR_INPUT
	ibGlobOff:	BOOL;
	ibGlobOffLong:	BOOL;
	irTemperature:	REAL;
	irHumidity:	REAL;
END_VAR
VAR PERSISTENT
	tyScene1: Type_SCENE_WZ;
	tyScene2: Type_SCENE_WZ;
	tyScene3: Type_SCENE_WZ;
	tyScene4: Type_SCENE_WZ;
	tyScene5: Type_SCENE_WZ;
	tyScene6: Type_SCENE_WZ;
	tyScene7: Type_SCENE_WZ;
	tyScene8: Type_SCENE_WZ;
	tyScene9: Type_SCENE_WZ;
	tyScene10: Type_SCENE_WZ;
	tyScene11: Type_SCENE_WZ;
	tyScene12: Type_SCENE_WZ;
	tyScene13: Type_SCENE_WZ;
	tyScene14: Type_SCENE_WZ;
	tyScene15: Type_SCENE_WZ;

	tyActScene:Type_SCENE_WZ;

	fbWhite:				PRG_FB_LED_SINGLE;
	fbRGBMirror1:		PRG_FB_LED_MULTI;
	fbRGBMirror2:		PRG_FB_LED_MULTI;
	fbRGBMirror3:		PRG_FB_LED_MULTI;
	fbWhiteTV:			PRG_FB_LED_SINGLE;

	fbPowerTV:PRG_FB_PULSE_SWITCH;
	SCENE_CONTROL:PRG_SCENE_CONTROL_WZ;
	nScene:INT;
	bLernen:BOOL;
	nBrightness:BYTE;
END_VAR
VAR_OUTPUT
	obDevOn:	BOOL;
END_VAR
(*Scene control*)
SCENE_CONTROL(
	i_bNextScene:= ,
	i_bPrevScene:= ,
	io_tyScene1:= tyScene1,
	io_tyScene2:= tyScene2,
	io_tyScene3:= tyScene3,
	io_tyScene4:= tyScene4,
	io_tyScene5:= tyScene5,
	io_tyScene6:= tyScene6,
	io_tyScene7:= tyScene7,
	io_tyScene8:= tyScene8,
	io_tyScene9:= tyScene9,
	io_tyScene10:= tyScene10,
	io_tyScene11:= tyScene11,
	io_tyScene12:= tyScene12,
	io_tyScene13:= tyScene13,
	io_tyScene14:= tyScene14,
	io_tyScene15:= tyScene15,
	o_tyActScene=> tyActScene,
	o_nScene => nScene);

(*LED light white*)
fbWhite(
	i_bSwitchOn:= FALSE,
	i_bSwitchOff:= ibGlobOff,
	i_bSwitchOnOff:= DI_S02_1,
	i_iSceneValue:= );

DO_S02_0 := fbWhite.bLight;

(*LED light RGB mirror 1*)
fbRGBMirror1(
	i_SwitchON:= FALSE,
	i_SwitchOFF:= ibGlobOff,
	i_bSwitchOnOff:= DI_S02_3,
	i_tyScene:= tyActScene.tyMirror1,
	i_nScene := nScene,
	di_SysTime:= di_System_Time);

(*LED light RGB mirror 2*)
fbRGBMirror2(
	i_SwitchON:= FALSE,
	i_SwitchOFF:= ibGlobOff,
	i_bSwitchOnOff:= DI_S02_3,
	i_tyScene:= tyActScene.tyMirror2,
	i_nScene := nScene,
	di_SysTime:= di_System_Time);

(*LED light RGB mirror 3*)
fbRGBMirror3(
	i_SwitchON:= FALSE,
	i_SwitchOFF:= ibGlobOff,
	i_bSwitchOnOff:= DI_S02_3,
	i_tyScene:= tyActScene.tyMirror3,
	i_nScene := nScene,
	di_SysTime:= di_System_Time);

(*relay for power supply*)
DO_NN_K03:=	fbWhite.bLight OR fbRGBMirror1.v_Type_LED_RGB.bLight OR fbRGBMirror2.v_Type_LED_RGB.bLight OR fbRGBMirror3.v_Type_LED_RGB.bLight;

DO_S02_0 := fbWhite.bLight;
DO_S02_2 :=  fbRGBMirror1.v_Type_LED_RGB.bLight OR fbRGBMirror1.v_Type_LED_RGB.bLight OR fbRGBMirror1.v_Type_LED_RGB.bLight;

(*relay for power supply TV*)
fbPowerTV(bTrigPlug:= DI_S02_5 OR (fbPowerTV.bStat AND ibGlobOffLong), bSwitchAck:= , bRelay=> DO_NN_K04);
DO_S02_4 := fbPowerTV.bStat OR (fbPowerPC.bStat OR fbPowerNAS.bStat OR fbPowerNasBackup.bStat) AND SYS_TOG_1S;

IF bLernen = TRUE THEN
	nBrightness := 0;
ELSE
	nBrightness := fbWhite.Brightness;
END_IF


(*DMX communication*)
arrDMXProcessData[20] := fbRGBMirror1.v_Type_LED_RGB.Red;
arrDMXProcessData[21] := fbRGBMirror1.v_Type_LED_RGB.Green;
arrDMXProcessData[22] := fbRGBMirror1.v_Type_LED_RGB.Blue;
arrDMXProcessData[23] := nBrightness;

arrDMXProcessData[30] := fbRGBMirror2.v_Type_LED_RGB.Red;
arrDMXProcessData[31] := fbRGBMirror2.v_Type_LED_RGB.Green;
arrDMXProcessData[32] := fbRGBMirror2.v_Type_LED_RGB.Blue;
arrDMXProcessData[33] :=  nBrightness;

arrDMXProcessData[40] := fbRGBMirror3.v_Type_LED_RGB.Red;
arrDMXProcessData[41] := fbRGBMirror3.v_Type_LED_RGB.Green;
arrDMXProcessData[42] := fbRGBMirror3.v_Type_LED_RGB.Blue;
arrDMXProcessData[43] := fbWhite.Brightness;


obDevOn:= 	fbWhite.bLight OR fbRGBMirror1.v_Type_LED_RGB.bLight OR fbRGBMirror2.v_Type_LED_RGB.bLight OR fbRGBMirror3.v_Type_LED_RGB.bLight OR
			fbPowerTV.bStat;
END_PROGRAM

(* POU Own PRG's and FB's/PRG_FB_LED_MULTI, ST *)
FUNCTION_BLOCK PRG_FB_LED_MULTI
VAR_INPUT
	i_SwitchON:	BOOL;
	i_SwitchOFF:	BOOL;
	i_bSwitchOnOff:	BOOL;
	i_nScene: INT;
	i_tyScene:	Type_LED_RGB;
	di_SysTime:	DINT;
END_VAR

VAR
	bDimmUp:			BOOL;
	bDimmDown:			BOOL;
	nDimmStep:			INT := 10;

	v_Type_LED_RGB: Type_LED_RGB;		(*CONTAINS THE LIGHT STATUS*)
	fnSwitchOnOff: F_TRIG;
	fpSwitchOnOff: R_TRIG;
	fnSwitchOn: F_TRIG;
	fnSwitchOff: F_TRIG;
	tiLongSwitchOnOff:	TON;
	tiLongSwitchOn:	TON;
	tiLongSwitchOff:	TON;
	fbDimmer2Switch: FB_Dimmer2Switch;
	fbContColor: PRG_CONT_COLOR;
	nScene:INT;
END_VAR
(*dimm up and down*)
bDimmUp := (tiLongSwitchOn.Q OR (tiLongSwitchOnOff.Q AND nDimmStep = 10)) AND NOT bDimmDown;
bDimmDown := (tiLongSwitchOff.Q OR (tiLongSwitchOnOff.Q AND nDimmStep = 20)) AND NOT bDimmUp;

(*flag negative edge and timer of switch for on*)
tiLongSwitchOn(IN:= i_SwitchON, PT:= T#500ms);
fnSwitchOn(CLK:= i_SwitchON );

(*flag negative edge and timer of switch for off*)
tiLongSwitchOff(IN:= i_SwitchOFF, PT:= T#500ms);
fnSwitchOff(CLK:= i_SwitchOFF );

(*flag negative edge and timer of switch for on and off*)
tiLongSwitchOnOff(IN:= i_bSwitchOnOff, PT:= T#500ms);
fnSwitchOnOff(CLK:= i_bSwitchOnOff );

(*nDimmStep = 20 ----> dimm down*)
IF tiLongSwitchOnOff.Q AND fbDimmer2Switch.nOut = 100  AND fpSwitchOnOff.Q THEN
	nDimmStep := 20;
END_IF

(*nDimmStep = 10 ----> dimm up*)
fpSwitchOnOff(CLK:= tiLongSwitchOnOff.Q );
IF tiLongSwitchOnOff.Q AND fbDimmer2Switch.nOut = 0 AND fpSwitchOnOff.Q THEN
	nDimmStep := 10;
END_IF

(*switch light on*)
IF fnSwitchOn.Q OR ( fnSwitchOnOff.Q AND NOT  v_Type_LED_RGB.bLight) THEN
(*IF i_SwitchON OR (v_Type_LED_RGB.fpSwitchOnOff.Q AND NOT v_Type_LED_RGB.bLight) THEN*)
	v_Type_LED_RGB.Switch_ON := TRUE;
END_IF

(*switch light off*)
IF (fnSwitchOff.Q AND NOT bDimmDown) OR ((fnSwitchOnOff.Q  AND NOT bDimmDown AND NOT bDimmUp) AND v_Type_LED_RGB.bLight) THEN
(*IF i_SwitchOFF OR (v_Type_LED_RGB.fpSwitchOnOff.Q AND v_Type_LED_RGB.bLight) THEN*)
	v_Type_LED_RGB.Switch_ON := FALSE;
END_IF

(*Scene has changed. Takeover new Scene*)
IF i_nScene <> nScene THEN
	nScene := i_nScene;
(*	v_Type_LED_RGB := i_tyScene;*)
	v_Type_LED_RGB.Config :=i_tyScene.Config;
	v_Type_LED_RGB.Hue :=i_tyScene.Hue;
	v_Type_LED_RGB.Saturation :=i_tyScene.Saturation;
	v_Type_LED_RGB.Switch_RANDOM :=i_tyScene.Switch_RANDOM;
END_IF

(*control light with standard FB from Beckhoff BaBasic Library*)
fbDimmer2Switch(
	bSwitchDimmUp:= bDimmUp,
	bSwitchDimmDown:= bDimmDown,
	bOn:= v_Type_LED_RGB.Switch_ON,
	bOff:= NOT v_Type_LED_RGB.Switch_ON,
	bSetDimmValue:= FALSE,
	nDimmValue:= 0,
	tSwitchOverTime:=T#300MS ,
	tDimmTime:= REAL_TO_TIME(v_Type_LED_RGB.Config.tDimmTime),
	bMemoryModeOn:= TRUE,
	nOnValueWithoutMemoryMode:= 0,
	bDimmOnMode:= v_Type_LED_RGB.Config.bDimmOnMode,
	tDimmOnTime:= REAL_TO_TIME(v_Type_LED_RGB.Config.tDimmOnTime),
	bDimmOffMode:= v_Type_LED_RGB.Config.bDimmOffMode,
	tDimmOffTime:= REAL_TO_TIME(v_Type_LED_RGB.Config.tDimmOffTime),
	nOutMin:= 0,
	nOutMax:=REAL_TO_UINT( v_Type_LED_RGB.Brightness),
	bLight=> v_Type_LED_RGB.bLight);

fbContColor(
	i_DimmValue:= fbDimmer2Switch.nOut,
	di_SysTime:= di_SysTime,
	io_Type_LED_RGB:= v_Type_LED_RGB );
END_FUNCTION_BLOCK

(* POU Own PRG's and FB's/PRG_CONT_COLOR, ST *)
FUNCTION_BLOCK PRG_CONT_COLOR
VAR_INPUT
	i_DimmValue:UINT;
	di_SysTime:	DINT;
END_VAR
VAR
	v_HUE: REAL;
	v_SATURATION: REAL;
	v_VALUE: REAL;
	v_VAR_H: REAL;
	v_VAR_I: REAL;
	v_VAR_1: REAL;
	v_VAR_2: REAL;
	v_VAR_3: REAL;
	v_VAR_R: REAL;
	v_VAR_G: REAL;
	v_VAR_B: REAL;
	v_Sys_Time_last_Call:	DINT;
	v_Cycle_Time:	DINT;
	v_RED: BYTE;
	v_GREEN: BYTE;
	v_BLUE: BYTE;
END_VAR

VAR_IN_OUT
	io_Type_LED_RGB: Type_LED_RGB;		(*CONTAINS THE LIGHT STATUS*)
END_VAR
(*Calculate the System Time between the last and the actual cycle for automatic color switching*)
v_Cycle_Time := di_SysTime - v_Sys_Time_last_Call;
v_Sys_Time_last_Call := di_SysTime;

IF io_Type_LED_RGB.Config.Speed_RANDOM < 1000 THEN
	io_Type_LED_RGB.Config.Speed_RANDOM := 1000;
END_IF

IF io_Type_LED_RGB.Switch_RANDOM AND io_Type_LED_RGB.Switch_ON THEN
	io_Type_LED_RGB.Hue := io_Type_LED_RGB.Hue + 360/(io_Type_LED_RGB.Config.Speed_RANDOM)*DINT_TO_REAL(v_Cycle_Time);

	IF io_Type_LED_RGB.Hue >= 360 THEN
		io_Type_LED_RGB.Hue := io_Type_LED_RGB.Hue-360;
	END_IF
	IF io_Type_LED_RGB.Hue < 0 THEN
		io_Type_LED_RGB.Hue := 0;
	END_IF
END_IF

v_HUE := io_Type_LED_RGB.Hue / 360;
v_SATURATION := io_Type_LED_RGB.Saturation / 100;
v_VALUE := (io_Type_LED_RGB.Brightness*UINT_TO_REAL(i_DimmValue)/100) / 100;

IF v_SATURATION = 0 THEN
	v_RED := REAL_TO_BYTE(v_VALUE * 255);
	v_GREEN := REAL_TO_BYTE(v_VALUE * 255);
	v_BLUE := REAL_TO_BYTE(v_VALUE * 255);
ELSE
	v_VAR_H := v_HUE * 6;
	v_VAR_I := FLOOR(REAL_TO_LREAL(v_VAR_H));
	v_VAR_1:= v_VALUE * (1 - v_SATURATION);
	v_VAR_2:= v_VALUE * (1 - v_SATURATION * (v_VAR_H - v_VAR_I));
	v_VAR_3:= v_VALUE * (1 - v_SATURATION * (1 - (v_VAR_H - v_VAR_I)));

	CASE REAL_TO_INT(v_VAR_I) OF
	0:
		v_VAR_R := v_VALUE;
		v_VAR_G := v_VAR_3;
		v_VAR_B := v_VAR_1;
	1:
		v_VAR_R := v_VAR_2;
		v_VAR_G := v_VALUE;
		v_VAR_B := v_VAR_1;
	2:
		v_VAR_R := v_VAR_1;
		v_VAR_G := v_VALUE;
		v_VAR_B := v_VAR_3;
	3:
		v_VAR_R := v_VAR_1;
		v_VAR_G := v_VAR_2;
		v_VAR_B := v_VALUE;
	4:
		v_VAR_R := v_VAR_3;
		v_VAR_G := v_VAR_1;
		v_VAR_B := v_VALUE;
	ELSE
		v_VAR_R := v_VALUE;
		v_VAR_G := v_VAR_1;
		v_VAR_B := v_VAR_2;
	END_CASE

	v_RED := REAL_TO_BYTE(v_VAR_R * 255);
	v_GREEN := REAL_TO_BYTE(v_VAR_G * 255);
	v_BLUE := REAL_TO_BYTE(v_VAR_B * 255);
END_IF


io_Type_LED_RGB.Red := v_RED;
io_Type_LED_RGB.Green := v_GREEN;
io_Type_LED_RGB.Blue := v_BLUE;
END_FUNCTION_BLOCK

(* POU Own PRG's and FB's/PRG_FB_PULSE_SWITCH, ST *)
FUNCTION_BLOCK PRG_FB_PULSE_SWITCH
VAR_INPUT
	bTrigOnOff:BOOL;
	bTrigPlug:BOOL;
	bSwitchAck:BOOL;
END_VAR
VAR_OUTPUT
	bRelay:BOOL;	(*digital output for relay*)
	bStat:BOOL;		(*status if pulse switch is on or off*)
END_VAR
VAR
	ftTrigPlug:F_TRIG;
	ftTrigOnOFF:F_TRIG;
	tonTrigPlug:TON;
	ftRelay:R_TRIG;
	fnRelay:F_TRIG;
	tofRelay:TOF;
END_VAR

VAR RETAIN
	bOn:BOOL;
END_VAR
ftTrigPlug(CLK:=bTrigPlug);
ftTrigOnOff(CLK:=bTrigOnOff);

IF (ftTrigOnOFF.Q OR (ftTrigPlug.Q AND NOT tonTrigPlug.Q) AND NOT  bStat) THEN
	 bOn := TRUE;
END_IF

IF (tonTrigPlug.Q OR ftTrigOnOFF.Q) AND bStat THEN
	 bOn := FALSE;
END_IF

ftRelay(CLK:= bOn);
fnRelay(CLK:=bOn);
tofRelay(IN:= ftRelay.Q OR fnRelay.Q, PT:=T#1s , Q=> bRelay);
bStat := bOn;

(*time must be at the end for correct function*)
tonTrigPlug(IN:=bTrigPlug , PT:=T#1s);
END_FUNCTION_BLOCK

(* POU Own PRG's and FB's/PRG_SCENE_CONTROL_WZ, ST *)
FUNCTION_BLOCK PRG_SCENE_CONTROL_WZ
VAR_INPUT
	i_bNextScene:	BOOL;
	i_bPrevScene:	BOOL;
END_VAR

VAR_IN_OUT
	io_tyScene1: Type_SCENE_WZ;
	io_tyScene2: Type_SCENE_WZ;
	io_tyScene3: Type_SCENE_WZ;
	io_tyScene4: Type_SCENE_WZ;
	io_tyScene5: Type_SCENE_WZ;
	io_tyScene6: Type_SCENE_WZ;
	io_tyScene7: Type_SCENE_WZ;
	io_tyScene8: Type_SCENE_WZ;
	io_tyScene9: Type_SCENE_WZ;
	io_tyScene10: Type_SCENE_WZ;
	io_tyScene11: Type_SCENE_WZ;
	io_tyScene12: Type_SCENE_WZ;
	io_tyScene13: Type_SCENE_WZ;
	io_tyScene14: Type_SCENE_WZ;
	io_tyScene15: Type_SCENE_WZ;
END_VAR

VAR_OUTPUT
	o_tyActScene: Type_SCENE_WZ;
	o_nScene:INT;
END_VAR

VAR
	fpNextScene: F_TRIG;
	fpPrevScene: F_TRIG;
	v_iActScene:	INT	:= 1;
END_VAR
fpNextScene(CLK:=i_bNextScene);
fpPrevScene(CLK:=i_bPrevScene);

IF fpNextScene.Q THEN
	v_iActScene := v_iActScene + 1;
END_IF

IF fpPrevScene.Q THEN
	v_iActScene := v_iActScene - 1;
END_IF

IF v_iActScene >= 17 THEN
	v_iActScene := 1;
END_IF

IF v_iActScene <= 0 THEN
	v_iActScene := 16;
END_IF

o_tyActScene := io_tyScene1;

CASE v_iActScene OF
1:	o_tyActScene := io_tyScene1;
2:	o_tyActScene := io_tyScene2;
3:	o_tyActScene := io_tyScene3;
4:	o_tyActScene := io_tyScene4;
5:	o_tyActScene := io_tyScene5;
6:	o_tyActScene := io_tyScene6;
7:	o_tyActScene := io_tyScene7;
8:	o_tyActScene := io_tyScene8;
9:	o_tyActScene := io_tyScene9;
10:	o_tyActScene := io_tyScene10;
11:	o_tyActScene := io_tyScene11;
12:	o_tyActScene := io_tyScene12;
13:	o_tyActScene := io_tyScene13;
14:	o_tyActScene := io_tyScene14;
15:	o_tyActScene := io_tyScene15;
END_CASE

o_nScene := v_iActScene;
END_FUNCTION_BLOCK

(* POU Rooms/ROOM_03_KUECHE, ST *)
PROGRAM ROOM_03_KUECHE
VAR_INPUT
	ibGlobOff:	BOOL;
	ibGlobOffLong:	BOOL;
	irTemperature:	REAL;
	irHumidity:	REAL;
END_VAR
VAR PERSISTENT
	fbWhiteCeiling: PRG_FB_LED_SINGLE;
END_VAR
VAR_OUTPUT
	obDevOn:	BOOL;
END_VAR
(*LED light white ceiling*)
fbWhiteCeiling(
	i_bSwitchOn:= FALSE,
	i_bSwitchOff:= ibGlobOff,
	i_bSwitchOnOff:=  DI_S03_1,
	i_iSceneValue:= );

(*relay for power supply*)
DO_NN_K05 :=	fbWhiteCeiling.bLight;


obDevOn:=	fbWhiteCeiling.bLight;
END_PROGRAM

(* POU Rooms/ROOM_04_ZIMMER, ST *)
PROGRAM ROOM_04_ZIMMER
VAR_INPUT
	ibGlobOff:	BOOL;
	ibGlobOffLong:	BOOL;
	irTemperature:	REAL;
	irHumidity:	REAL;
	irTemperatureSZ:	REAL;
	irHumiditySZ:	REAL;
END_VAR
VAR PERSISTENT
	fbWhiteCeiling:			PRG_FB_LED_SINGLE;
	fbWhiteSZCeiling:			PRG_FB_LED_SINGLE;
	fbWhiteSZReadLeft:		PRG_FB_LED_SINGLE;
	fbWhiteSZReadRight:		PRG_FB_LED_SINGLE;
END_VAR
VAR
	fnNightModeOn:F_TRIG;
	fnNightModeOff:F_TRIG;
	tNightMode: TON;
	tLightAutoSwitchOff: TON;
	fpLightAutoSwitchOff:R_TRIG;

	fnLightBed: F_TRIG;
END_VAR
VAR_OUTPUT
	obDevOn:	BOOL;
END_VAR
(*LED light white ceiling*)
fbWhiteCeiling(
	i_bSwitchOn:= FALSE,
	i_bSwitchOff:= FALSE,
	i_bSwitchOnOff:= DI_S04_2,
	i_iSceneValue:= );

(*LED light white SZ ceiling*)
fbWhiteSZCeiling(
	i_bSwitchOn:= FALSE,
	i_bSwitchOff:= ibGlobOff OR fpLightAutoSwitchOff.Q,
	i_bSwitchOnOff:= DI_S05_1 OR DI_S06_2 OR DI_S07_2,
	i_iSceneValue:= );

DO_S05_0 := fbWhiteSZCeiling.bLight;
DO_S06_1 := fbWhiteSZCeiling.bLight;

(*Nachtmodus automatisch um 22 Uhr einschalten und um 6 Uhr ausschalten*)
fnNightModeOn(CLK:= NOT bNightMode AND (DI_S05_4 OR DI_S06_4 OR  (fbTime.systemTime.wHour = 21 AND fbTime.systemTime.wMinute = 59)));
fnNightModeOff(CLK:= bNightMode AND (DI_S05_4 OR DI_S06_4  OR  (fbTime.systemTime.wHour = 6 AND fbTime.systemTime.wMinute = 59)));

IF fnNightModeOn.Q THEN
	bNightMode := TRUE;
END_IF

IF fnNightModeOff.Q THEN
	bNightMode := FALSE;
END_IF

(*Lich nach 15 Minuten ausschalten*)
tLightAutoSwitchOff(IN:=fbWhiteSZCeiling.bLight OR fbWhiteSZReadLeft.bLight OR fbWhiteSZReadRight.bLight, PT:= T#15M );
fpLightAutoSwitchOff(CLK:=tLightAutoSwitchOff.Q);

fnLightBed(CLK:= DI_S07_1);

(*LED light white SZ read left*)
fbWhiteSZReadLeft(
	i_bSwitchOn:= FALSE,
	i_bSwitchOff:= ibGlobOff OR fpLightAutoSwitchOff.Q OR (fnLightBed.Q AND (fbWhiteSZReadRight.bLight <> fbWhiteSZReadLeft.bLight)),
	i_bSwitchOnOff:= DI_S05_2 OR (fnLightBed.Q AND (fbWhiteSZReadRight.bLight = fbWhiteSZReadLeft.bLight)),
	i_iSceneValue:= );

DO_S05_1 := fbWhiteSZReadLeft.bLight;

(*LED light white SZ read right*)
fbWhiteSZReadRight(
	i_bSwitchOn:= FALSE,
	i_bSwitchOff:= ibGlobOff OR fpLightAutoSwitchOff.Q OR (fnLightBed.Q AND (fbWhiteSZReadRight.bLight <> fbWhiteSZReadLeft.bLight)),
	i_bSwitchOnOff:= DI_S06_1 OR (fnLightBed.Q AND (fbWhiteSZReadRight.bLight = fbWhiteSZReadLeft.bLight)),
	i_iSceneValue:= );

DO_S06_0 := fbWhiteSZReadRight.bLight;



(*relay for power supply*)
DO_NN_K06 :=	fbWhiteCeiling.bLight OR fbWhiteSZCeiling.bLight OR fbWhiteSZReadLeft.bLight OR fbWhiteSZReadRight.bLight;

(*DMX communication*)
arrDMXProcessData[50] := fbWhiteCeiling.Brightness;
arrDMXProcessData[51] := fbWhiteSZCeiling.Brightness;
arrDMXProcessData[52] := fbWhiteSZReadLeft.Brightness;
arrDMXProcessData[53] := fbWhiteSZReadRight.Brightness;

obDevOn:=	fbWhiteCeiling.bLight OR fbWhiteSZCeiling.bLight OR fbWhiteSZReadLeft.bLight OR fbWhiteSZReadRight.bLight;
END_PROGRAM

(* POU Rooms/ROOM_05_WC_GANG, ST *)
PROGRAM ROOM_05_WC_GANG
VAR_INPUT
	ibGlobOff:	BOOL;
	ibGlobOffLong:	BOOL;
END_VAR
VAR PERSISTENT
	fbWhiteWC:			PRG_FB_LED_SINGLE;
	fbWhiteGarderobe:	PRG_FB_LED_SINGLE;
	fbWhiteAreaKitchen:	PRG_FB_LED_SINGLE;
	fbWhiteBalkon:		PRG_FB_LED_SINGLE;

	bWhiteGangEin: BOOL;
	baxWhiteGangEin: BOOL;
	fnWhiteGangEin: F_TRIG;

	nTest: BYTE;
	nBrightnessNightMode:INT;
END_VAR
VAR
	fbLightBathroom: FB_Light;

	fpBM2:R_TRIG;
	fnBM2:F_TRIG;
	tDoffBM2: TOF;
	fpBM3:R_TRIG;
	fnBM3:F_TRIG;
	tDoffBM3: TOF;
	tDonVentWC: TON;
	tDoffVentWC: TOF;
	tWCLightAutoSwitchOff: TON;
	fpWCLightAutoSwitchOff: R_TRIG;
	tGangLightAutoSwitchOff: TON;
	fpGangLightAutoSwitchOff: R_TRIG;

END_VAR
VAR_OUTPUT
	obDevOn:	BOOL;
END_VAR
tWCLightAutoSwitchOff(IN:=fbWhiteWC.bLight, PT:= T#15M);
fpWCLightAutoSwitchOff(CLK:=tWCLightAutoSwitchOff.Q);

(*LED light white WC*)
fbWhiteWC(
	i_bSwitchOn:= FALSE,
	i_bSwitchOff:= fpWCLightAutoSwitchOff.Q,
	i_bSwitchOnOff:= DI_S08,
	i_iSceneValue:= );


tDoffVentWC(IN:= (tDonVentWC.Q AND NOT fbWhiteWC.bLight), PT:= T#2m, Q=> DO_NN_K09);
tDonVentWC(IN:= fbWhiteWC.bLight, PT:=T#2m );

(*flags of BM*)
tDoffBM2(IN:= DI_BM2, PT:= T#1s);
tDoffBM3(IN:= DI_BM3, PT:= T#1s);

fpBM2(CLK:= tDoffBM2.Q);
fnBM2(CLK:= tDoffBM2.Q);
fpBM3(CLK:= tDoffBM3.Q);
fnBM3(CLK:= tDoffBM3.Q);

fnWhiteGangEin(CLK:= DI_S03_2);

IF fnWhiteGangEin.Q AND NOT baxWhiteGangEin THEN
	bWhiteGangEin := TRUE;
END_IF

IF (fnWhiteGangEin.Q OR fpGangLightAutoSwitchOff.Q) AND  baxWhiteGangEin THEN
	bWhiteGangEin := FALSE;
END_IF

baxWhiteGangEin := bWhiteGangEin;

tGangLightAutoSwitchOff(IN:=(fbWhiteGarderobe.bLight OR fbWhiteAreaKitchen.bLight) AND bWhiteGangEin, PT:= T#60M);
fpGangLightAutoSwitchOff(CLK:=tGangLightAutoSwitchOff.Q);

(*LED light white*)
fbWhiteGarderobe(
	i_bSwitchOn:= ((fpBM2.Q AND NOT bWhiteGangEin) OR (bWhiteGangEin AND fnWhiteGangEin.Q AND NOT fbWhiteGarderobe.bLight)),
	i_bSwitchOff:= (fnBM2.Q AND NOT bWhiteGangEin) OR (NOT bWhiteGangEin AND fnWhiteGangEin.Q AND fbWhiteGarderobe.bLight) OR fpGangLightAutoSwitchOff.Q,
	i_bSwitchOnOff:= FALSE,
	i_iSceneValue:= );

(*LED light white*)
fbWhiteAreaKitchen(
	i_bSwitchOn:= ((fpBM3.Q AND NOT bWhiteGangEin) OR (bWhiteGangEin AND fnWhiteGangEin.Q AND NOT fbWhiteAreaKitchen.bLight)),
	i_bSwitchOff:= (fnBM3.Q AND NOT bWhiteGangEin) OR (NOT bWhiteGangEin AND fnWhiteGangEin.Q AND fbWhiteAreaKitchen.bLight) OR fpGangLightAutoSwitchOff.Q,
	i_bSwitchOnOff:= FALSE,
	i_iSceneValue:= );

(*LED light white*)
fbWhiteBalkon(
	i_bSwitchOn:= FALSE,
	i_bSwitchOff:= ibGlobOff,
	i_bSwitchOnOff:= DI_S02_4,
	i_iSceneValue:= );

DO_S02_3 := fbWhiteBalkon.bLight;

(*relay for power supply*)
DO_NN_K07 :=	fbWhiteWC.bLight OR fbWhiteGarderobe.bLight OR fbWhiteAreaKitchen.bLight OR fbWhiteBalkon.bLight;

(*light bathroom*)
fbLightBathroom(bOn:=FALSE , bOff:=FALSE , bToggle:=DI_S11 , bLight=> DO_NN_K08);


IF bNightMode THEN
	nBrightnessNightMode := 100;
ELSE
	nBrightnessNightMode := 255;
END_IF

(*DMX communication*)

arrDMXProcessData[60] :=  INT_TO_BYTE(PRG_MAX_BRIGHTNESS(fbWhiteAreaKitchen.Brightness, 0, nBrightnessNightMode));
arrDMXProcessData[61] := INT_TO_BYTE(PRG_MAX_BRIGHTNESS(fbWhiteGarderobe.Brightness, 0, nBrightnessNightMode));
arrDMXProcessData[62] := INT_TO_BYTE(PRG_MAX_BRIGHTNESS(fbWhiteWC.Brightness, 0, nBrightnessNightMode));
arrDMXProcessData[63] :=fbWhiteBalkon.Brightness;


obDevOn:=	fbWhiteWC.bLight OR fbWhiteGarderobe.bLight OR fbWhiteAreaKitchen.bLight OR fbWhiteBalkon.bLight OR fbLightBathroom.bLight;
END_PROGRAM

(* POU Own PRG's and FB's/PRG_MAX_BRIGHTNESS, ST *)
FUNCTION PRG_MAX_BRIGHTNESS : INT
VAR_INPUT
	nBYTE:INT;
	nMin:INT;
	nMax:INT;
END_VAR
VAR
END_VAR
IF nBYTE < nMin THEN
	PRG_MAX_BRIGHTNESS:=nMIN;
ELSE IF nBYTE > nMAX THEN
	PRG_MAX_BRIGHTNESS:=nMAX;
ELSE
	PRG_MAX_BRIGHTNESS:=nBYTE;
END_IF;
END_IF;
END_FUNCTION

(* POU General/SYS_01_TREND, ST *)
PROGRAM SYS_01_TREND
VAR_INPUT
	irTemperatureSchlafzimmer:	REAL;
	irHumiditySchlafzimmer:	REAL;
	irTemperatureKinderzimmer:	REAL;
	irHumidityKinderzimmer:	REAL;
	irTemperatureKueche:	REAL;
	irHumidityKueche:	REAL;
	irTemperatureTerrariumLinks:	REAL;
	irHumidityTerrariumLinks:	REAL;
	irTemperatureTerrariumRechts:	REAL;
	irHumidityTerrariumRechts:	REAL;
END_VAR
VAR
	nActSensorNumber:INT:=1;
	nMaxSensorNumber:INT:=10;
	bRSTFifo:BOOL;
	fpMinute:R_TRIG;
	eState: E_SQLStatement;

	NT_GetTime1: NT_GetTime;
	bTimestart:BOOL;
	tTime: TIMESTRUCT;

        FB_FormatString1: FB_FormatString;
        sInsertString: T_MaxString;
        bError: BOOL;
        nErrid: UDINT;

        FB_DBRecordInsert1: FB_DBRecordInsert;
        bBusyInsert: BOOL;
        bErrInsert: BOOL;
        nErridInsert: UDINT;
        stSQLStateInsert: ST_DBSQLError;

	tStartInput:TON;
	bBusy:BOOL;
	fneRecordInsertFinished:F_TRIG;
END_VAR
(*Create the timestamp*)
NT_GetTime1( START:= bTimestart, TIMESTR=> tTime);
IF NOT NT_GetTime1.BUSY THEN
	bTimestart := NOT bTimestart;
END_IF

fpMinute(CLK:= (tTime.wSecond=0) );

IF fpMinute.Q THEN

	(*Write Value into FIFO*)
	TemperatureSchlafzimmerFIFO(
		REALin:= irTemperatureSchlafzimmer,
		tTime:= tTime,
		E:=TRUE ,
		RD:= FALSE,
		WD:=fpMinute.Q,
		RST:= bRSTFifo  );

	(*Write Value into FIFO*)
	HumiditySchlafzimmerFIFO(
		REALin:= irHumiditySchlafzimmer,
		tTime:= tTime,
		E:=TRUE ,
		RD:= FALSE,
		WD:=fpMinute.Q,
		RST:= bRSTFifo  );

	(*Write Value into FIFO*)
	TemperatureKinderzimmerFIFO(
		REALin:= irTemperatureKinderzimmer,
		tTime:= tTime,
		E:=TRUE ,
		RD:= FALSE,
		WD:=fpMinute.Q,
		RST:= bRSTFifo  );

	(*Write Value into FIFO*)
	HumidityKinderzimmerFIFO(
		REALin:= irHumidityKinderzimmer,
		tTime:= tTime,
		E:=TRUE ,
		RD:= FALSE,
		WD:=fpMinute.Q,
		RST:= bRSTFifo  );

	(*Write Value into FIFO*)
	TemperatureKuecheFIFO(
		REALin:= irTemperatureKueche,
		tTime:= tTime,
		E:=TRUE ,
		RD:= FALSE,
		WD:=fpMinute.Q,
		RST:=  bRSTFifo );

	(*Write Value into FIFO*)
	HumidityKuecheFIFO(
		REALin:= irHumidityKueche,
		tTime:= tTime,
		E:=TRUE ,
		RD:= FALSE,
		WD:=fpMinute.Q,
		RST:= bRSTFifo  );

	(*Write Value into FIFO*)
	TemperatureTerrariumLinksFIFO(
		REALin:= irTemperatureTerrariumLinks,
		tTime:= tTime,
		E:=TRUE ,
		RD:= FALSE,
		WD:=fpMinute.Q,
		RST:= bRSTFifo  );

	(*Write Value into FIFO*)
	HumidityTerrariumLinksFIFO(
		REALin:= irHumidityTerrariumLinks,
		tTime:= tTime,
		E:=TRUE ,
		RD:= FALSE,
		WD:=fpMinute.Q,
		RST:= bRSTFifo  );

	(*Write Value into FIFO*)
	TemperatureTerrariumRechtsFIFO(
		REALin:= irTemperatureTerrariumRechts,
		tTime:= tTime,
		E:=TRUE ,
		RD:= FALSE,
		WD:=fpMinute.Q,
		RST:= bRSTFifo  );

	(*Write Value into FIFO*)
	HumidityTerrariumRechtsFIFO(
		REALin:= irHumidityTerrariumRechts,
		tTime:= tTime,
		E:=TRUE ,
		RD:= FALSE,
		WD:=fpMinute.Q,
		RST:= bRSTFifo  );

END_IF



CASE nActSensorNumber OF
	1:	 (*Create the SQL-INSERT command*)
                	FB_FormatString1(
                        sFormat:= 'INSERT INTO myHome (timestamp, varname, value) VALUES ($'%D-%D-%D %D:%D:00$',$'%S$',$'%F$')',
                        arg1:= F_WORD(TemperatureSchlafzimmerFIFO.YEARout),
                        arg2:= F_WORD(TemperatureSchlafzimmerFIFO.MONTHout),
                        arg3:= F_WORD(TemperatureSchlafzimmerFIFO.DAYout),
                        arg4:= F_WORD(TemperatureSchlafzimmerFIFO.HOURout),
		     arg5:= F_WORD(TemperatureSchlafzimmerFIFO.MINUTEout),
                        arg6:= F_STRING('Temperatur Schlafzimmer'),
		     arg7:= F_REAL(TemperatureSchlafzimmerFIFO.REALout),
                        sOut=> sInsertString,
                        bError=> bError,
                        nErrId=> nErrid);

		IF NOT TemperatureSchlafzimmerFIFO.EMPTY THEN
			tStartInput(IN:=NOT FB_DBRecordInsert1.bBusy , PT:= T#200ms);
		END_IF

		IF  TemperatureSchlafzimmerFIFO.EMPTY THEN
			nActSensorNumber:=nActSensorNumber+1;
		END_IF

		IF fneRecordInsertFinished.Q AND NOT bErrInsert THEN
			TemperatureSchlafzimmerFIFO(
				E:=TRUE ,
				RD:=TRUE,
				WD:=FALSE);
			tStartInput(IN:=FALSE);
			nActSensorNumber:=nActSensorNumber+1;
		END_IF

	2:	 (*Create the SQL-INSERT command*)
                	FB_FormatString1(
                        sFormat:= 'INSERT INTO myHome (timestamp, varname, value) VALUES ($'%D-%D-%D %D:%D:00$',$'%S$',$'%F$')',
                        arg1:= F_WORD(HumiditySchlafzimmerFIFO.YEARout),
                        arg2:= F_WORD(HumiditySchlafzimmerFIFO.MONTHout),
                        arg3:= F_WORD(HumiditySchlafzimmerFIFO.DAYout),
                        arg4:= F_WORD(HumiditySchlafzimmerFIFO.HOURout),
		     arg5:= F_WORD(HumiditySchlafzimmerFIFO.MINUTEout),
                        arg6:= F_STRING('Feuchtigkeit Schlafzimmer'),
		     arg7:= F_REAL(HumiditySchlafzimmerFIFO.REALout),
                        sOut=> sInsertString,
                        bError=> bError,
                        nErrId=> nErrid);

		IF NOT HumiditySchlafzimmerFIFO.EMPTY  THEN
			tStartInput(IN:=NOT FB_DBRecordInsert1.bBusy , PT:= T#200ms);
		END_IF

		IF  HumiditySchlafzimmerFIFO.EMPTY THEN
			nActSensorNumber:=nActSensorNumber+1;
		END_IF

		IF fneRecordInsertFinished.Q AND NOT bErrInsert THEN
			HumiditySchlafzimmerFIFO(
				E:=TRUE ,
				RD:=TRUE,
				WD:=FALSE);
			tStartInput(IN:=FALSE);
			nActSensorNumber:=nActSensorNumber+1;
		END_IF


	3:	 (*Create the SQL-INSERT command*)
                	FB_FormatString1(
                        sFormat:= 'INSERT INTO myHome (timestamp, varname, value) VALUES ($'%D-%D-%D %D:%D:00$',$'%S$',$'%F$')',
                        arg1:= F_WORD(TemperatureKinderzimmerFIFO.YEARout),
                        arg2:= F_WORD(TemperatureKinderzimmerFIFO.MONTHout),
                        arg3:= F_WORD(TemperatureKinderzimmerFIFO.DAYout),
                        arg4:= F_WORD(TemperatureKinderzimmerFIFO.HOURout),
		     arg5:= F_WORD(TemperatureKinderzimmerFIFO.MINUTEout),
                        arg6:= F_STRING('Temperatur Kinderzimmer'),
		     arg7:= F_REAL(TemperatureKinderzimmerFIFO.REALout),
                        sOut=> sInsertString,
                        bError=> bError,
                        nErrId=> nErrid);

		IF NOT TemperatureKinderzimmerFIFO.EMPTY  THEN
			tStartInput(IN:=NOT FB_DBRecordInsert1.bBusy , PT:= T#200ms);
		END_IF

		IF  TemperatureKinderzimmerFIFO.EMPTY THEN
			nActSensorNumber:=nActSensorNumber+1;
		END_IF

		IF fneRecordInsertFinished.Q AND NOT bErrInsert THEN
			TemperatureKinderzimmerFIFO(
				E:=TRUE ,
				RD:=TRUE,
				WD:=FALSE);
			tStartInput(IN:=FALSE);
			nActSensorNumber:=nActSensorNumber+1;
		END_IF


	4:	 (*Create the SQL-INSERT command*)
                	FB_FormatString1(
                        sFormat:= 'INSERT INTO myHome (timestamp, varname, value) VALUES ($'%D-%D-%D %D:%D:00$',$'%S$',$'%F$')',
                        arg1:= F_WORD(HumidityKinderzimmerFIFO.YEARout),
                        arg2:= F_WORD(HumidityKinderzimmerFIFO.MONTHout),
                        arg3:= F_WORD(HumidityKinderzimmerFIFO.DAYout),
                        arg4:= F_WORD(HumidityKinderzimmerFIFO.HOURout),
		     arg5:= F_WORD(HumidityKinderzimmerFIFO.MINUTEout),
                        arg6:= F_STRING('Feuchtigkeit Kinderzimmer'),
		     arg7:= F_REAL(HumidityKinderzimmerFIFO.REALout),
                        sOut=> sInsertString,
                        bError=> bError,
                        nErrId=> nErrid);

		IF NOT HumidityKinderzimmerFIFO.EMPTY  THEN
			tStartInput(IN:=NOT FB_DBRecordInsert1.bBusy , PT:= T#200ms);
		END_IF

		IF  HumidityKinderzimmerFIFO.EMPTY THEN
			nActSensorNumber:=nActSensorNumber+1;
		END_IF

		IF fneRecordInsertFinished.Q AND NOT bErrInsert THEN
			HumidityKinderzimmerFIFO(
				E:=TRUE ,
				RD:=TRUE,
				WD:=FALSE);
			tStartInput(IN:=FALSE);
			nActSensorNumber:=nActSensorNumber+1;
		END_IF


	5:	 (*Create the SQL-INSERT command*)
                	FB_FormatString1(
                        sFormat:= 'INSERT INTO myHome (timestamp, varname, value) VALUES ($'%D-%D-%D %D:%D:00$',$'%S$',$'%F$')',
                        arg1:= F_WORD(TemperatureKuecheFIFO.YEARout),
                        arg2:= F_WORD(TemperatureKuecheFIFO.MONTHout),
                        arg3:= F_WORD(TemperatureKuecheFIFO.DAYout),
                        arg4:= F_WORD(TemperatureKuecheFIFO.HOURout),
		     arg5:= F_WORD(TemperatureKuecheFIFO.MINUTEout),
                        arg6:= F_STRING('Temperatur Kueche'),
		     arg7:= F_REAL(TemperatureKuecheFIFO.REALout),
                        sOut=> sInsertString,
                        bError=> bError,
                        nErrId=> nErrid);

		IF NOT TemperatureKuecheFIFO.EMPTY THEN
			tStartInput(IN:=NOT FB_DBRecordInsert1.bBusy , PT:= T#200ms);
		END_IF

		IF  TemperatureKuecheFIFO.EMPTY THEN
			nActSensorNumber:=nActSensorNumber+1;
		END_IF

		IF fneRecordInsertFinished.Q AND NOT bErrInsert THEN
			TemperatureKuecheFIFO(
				E:=TRUE ,
				RD:=TRUE,
				WD:=FALSE);
			tStartInput(IN:=FALSE);
			nActSensorNumber:=nActSensorNumber+1;
		END_IF


	6:	 (*Create the SQL-INSERT command*)
                	FB_FormatString1(
                        sFormat:= 'INSERT INTO myHome (timestamp, varname, value) VALUES ($'%D-%D-%D %D:%D:00$',$'%S$',$'%F$')',
                        arg1:= F_WORD(HumidityKuecheFIFO.YEARout),
                        arg2:= F_WORD(HumidityKuecheFIFO.MONTHout),
                        arg3:= F_WORD(HumidityKuecheFIFO.DAYout),
                        arg4:= F_WORD(HumidityKuecheFIFO.HOURout),
		     arg5:= F_WORD(HumidityKuecheFIFO.MINUTEout),
                        arg6:= F_STRING('Feuchtigkeit Kueche'),
		     arg7:= F_REAL(HumidityKuecheFIFO.REALout),
                        sOut=> sInsertString,
                        bError=> bError,
                        nErrId=> nErrid);

		IF NOT HumidityKuecheFIFO.EMPTY  THEN
			tStartInput(IN:=NOT FB_DBRecordInsert1.bBusy , PT:= T#200ms);
		END_IF

		IF  HumidityKuecheFIFO.EMPTY THEN
			nActSensorNumber:=nActSensorNumber+1;
		END_IF

		IF fneRecordInsertFinished.Q AND NOT bErrInsert THEN
			HumidityKuecheFIFO(
				E:=TRUE ,
				RD:=TRUE,
				WD:=FALSE);
			tStartInput(IN:=FALSE);
			nActSensorNumber:=nActSensorNumber+1;
		END_IF

	7:	 (*Create the SQL-INSERT command*)
                	FB_FormatString1(
                        sFormat:= 'INSERT INTO myHome (timestamp, varname, value) VALUES ($'%D-%D-%D %D:%D:00$',$'%S$',$'%F$')',
                        arg1:= F_WORD(TemperatureTerrariumLinksFIFO.YEARout),
                        arg2:= F_WORD(TemperatureTerrariumLinksFIFO.MONTHout),
                        arg3:= F_WORD(TemperatureTerrariumLinksFIFO.DAYout),
                        arg4:= F_WORD(TemperatureTerrariumLinksFIFO.HOURout),
		     arg5:= F_WORD(TemperatureTerrariumLinksFIFO.MINUTEout),
                        arg6:= F_STRING('Temperatur Terrarium Links'),
		     arg7:= F_REAL(TemperatureTerrariumLinksFIFO.REALout),
                        sOut=> sInsertString,
                        bError=> bError,
                        nErrId=> nErrid);

		IF NOT TemperatureTerrariumLinksFIFO.EMPTY  THEN
			tStartInput(IN:=NOT FB_DBRecordInsert1.bBusy , PT:= T#200ms);
		END_IF

		IF  TemperatureTerrariumLinksFIFO.EMPTY THEN
			nActSensorNumber:=nActSensorNumber+1;
		END_IF

		IF fneRecordInsertFinished.Q AND NOT bErrInsert THEN
			TemperatureTerrariumLinksFIFO(
				E:=TRUE ,
				RD:=TRUE,
				WD:=FALSE);
			tStartInput(IN:=FALSE);
			nActSensorNumber:=nActSensorNumber+1;
		END_IF

	8:	 (*Create the SQL-INSERT command*)
                	FB_FormatString1(
                        sFormat:= 'INSERT INTO myHome (timestamp, varname, value) VALUES ($'%D-%D-%D %D:%D:00$',$'%S$',$'%F$')',
                        arg1:= F_WORD(HumidityTerrariumLinksFIFO.YEARout),
                        arg2:= F_WORD(HumidityTerrariumLinksFIFO.MONTHout),
                        arg3:= F_WORD(HumidityTerrariumLinksFIFO.DAYout),
                        arg4:= F_WORD(HumidityTerrariumLinksFIFO.HOURout),
		     arg5:= F_WORD(HumidityTerrariumLinksFIFO.MINUTEout),
                        arg6:= F_STRING('Feuchtigkeit Terrarium Links'),
		     arg7:= F_REAL(HumidityTerrariumLinksFIFO.REALout),
                        sOut=> sInsertString,
                        bError=> bError,
                        nErrId=> nErrid);

		IF NOT HumidityTerrariumLinksFIFO.EMPTY  THEN
			tStartInput(IN:=NOT FB_DBRecordInsert1.bBusy , PT:= T#200ms);
		END_IF

		IF  HumidityTerrariumLinksFIFO.EMPTY THEN
			nActSensorNumber:=nActSensorNumber+1;
		END_IF

		IF fneRecordInsertFinished.Q AND NOT bErrInsert THEN
			HumidityTerrariumLinksFIFO(
				E:=TRUE ,
				RD:=TRUE,
				WD:=FALSE);
			tStartInput(IN:=FALSE);
			nActSensorNumber:=nActSensorNumber+1;
		END_IF

	9:	 (*Create the SQL-INSERT command*)
                	FB_FormatString1(
                        sFormat:= 'INSERT INTO myHome (timestamp, varname, value) VALUES ($'%D-%D-%D %D:%D:00$',$'%S$',$'%F$')',
                        arg1:= F_WORD(TemperatureTerrariumRechtsFIFO.YEARout),
                        arg2:= F_WORD(TemperatureTerrariumRechtsFIFO.MONTHout),
                        arg3:= F_WORD(TemperatureTerrariumRechtsFIFO.DAYout),
                        arg4:= F_WORD(TemperatureTerrariumRechtsFIFO.HOURout),
		     arg5:= F_WORD(TemperatureTerrariumRechtsFIFO.MINUTEout),
                        arg6:= F_STRING('Temperatur Terrarium Rechts'),
		     arg7:= F_REAL(TemperatureTerrariumRechtsFIFO.REALout),
                        sOut=> sInsertString,
                        bError=> bError,
                        nErrId=> nErrid);

		IF NOT TemperatureTerrariumRechtsFIFO.EMPTY  THEN
			tStartInput(IN:=NOT FB_DBRecordInsert1.bBusy , PT:= T#200ms);
		END_IF

		IF  TemperatureTerrariumRechtsFIFO.EMPTY THEN
			nActSensorNumber:=nActSensorNumber+1;
		END_IF

		IF fneRecordInsertFinished.Q AND NOT bErrInsert THEN
			TemperatureTerrariumRechtsFIFO(
				E:=TRUE ,
				RD:=TRUE,
				WD:=FALSE);
			tStartInput(IN:=FALSE);
			nActSensorNumber:=nActSensorNumber+1;
		END_IF

	10:	 (*Create the SQL-INSERT command*)
                	FB_FormatString1(
                        sFormat:= 'INSERT INTO myHome (timestamp, varname, value) VALUES ($'%D-%D-%D %D:%D:00$',$'%S$',$'%F$')',
                        arg1:= F_WORD(HumidityTerrariumRechtsFIFO.YEARout),
                        arg2:= F_WORD(HumidityTerrariumRechtsFIFO.MONTHout),
                        arg3:= F_WORD(HumidityTerrariumRechtsFIFO.DAYout),
                        arg4:= F_WORD(HumidityTerrariumRechtsFIFO.HOURout),
		     arg5:= F_WORD(HumidityTerrariumRechtsFIFO.MINUTEout),
                        arg6:= F_STRING('Feuchtigkeit Terrarium Rechts'),
		     arg7:= F_REAL(HumidityTerrariumRechtsFIFO.REALout),
                        sOut=> sInsertString,
                        bError=> bError,
                        nErrId=> nErrid);

		IF NOT HumidityTerrariumRechtsFIFO.EMPTY  THEN
			tStartInput(IN:=NOT FB_DBRecordInsert1.bBusy , PT:= T#200ms);
		END_IF

		IF  HumidityTerrariumRechtsFIFO.EMPTY THEN
			nActSensorNumber:=nActSensorNumber+1;
		END_IF

		IF fneRecordInsertFinished.Q AND NOT bErrInsert THEN
			HumidityTerrariumRechtsFIFO(
				E:=TRUE ,
				RD:=TRUE,
				WD:=FALSE);
			tStartInput(IN:=FALSE);
			nActSensorNumber:=nActSensorNumber+1;
		END_IF
END_CASE

          (*-------------------------------------------------------------------------*)

                (*Write the record to the database*)
                FB_DBRecordInsert1(
                        sNetID:= ,
                        hDBID:= 1,
                        sInsertCmd:= sInsertString,
                        bExecute:= tStartInput.Q,
                        tTimeout:= T#15s,
                        bBusy=> bBusyInsert,
                        bError=> bErrInsert,
                        nErrID=> nErridInsert,
                        sSQLState=> stSQLStateInsert);


fneRecordInsertFinished(CLK:= bBusyInsert);


IF nActSensorNumber > nMaxSensorNumber THEN
	nActSensorNumber:=1;
END_IF
END_PROGRAM

(* POU FAST, ST *)
PROGRAM FAST
VAR
	(* background communication with the COM port device *)
	COMportControl: SerialLineControl;
	COMportControlError: BOOL;
	COMportControlErrorID: ComError_t;

END_VAR
(*==================================================================
	Background communication with KL6001 terminal
	The SerialLineControl function block is supposed to be called in every PLC cycle.
	It communicates with the serial line hardware device and transmits or receives data.
	The SerialLineControl can be called in the standard task or in a separate fast task as well.
	A fast separate task will be necessary at high baud rates or 
	with KL6001 terminals which have a small process image (3 or 5 data bytes only)
*)
COMportControl(
	Mode:= SERIALLINEMODE_KL6_22B_STANDARD,
	pComIn:= ADR(COMin_KL6001),			(* I/O data; see global variables *)
	pComOut:= ADR(COMout_KL6001),		(* I/O data; see global variables *)
	SizeComIn:= SIZEOF(COMin_KL6001),	(* I/O data; see global variables *)
	TxBuffer:= TxBuffer2,				(* transmit buffer; see global variables *)
	RxBuffer:= RxBuffer2,				(* receive buffer; see global variables *)
	Error=> COMportControlError,
	ErrorID=> COMportControlErrorID );
END_PROGRAM

(* POU Own PRG's and FB's/PRG_LED_SINGLECOLOR, ST *)
PROGRAM PRG_LED_SINGLECOLOR
VAR_INPUT
	i_bSwitchOn:		BOOL;
	i_bSwitchOff:		BOOL;
	i_bSwitchOnOff:	BOOL;
	i_iSceneValue:	INT;
END_VAR

VAR_IN_OUT
	io_TypeLED: Type_LED;		(*CONTAINS THE LIGHT STATUS*)
END_VAR
(*flag positive edge of switch for on and off*)
io_TypeLED.fpSwitchOnOff(CLK:= i_bSwitchOnOff );

(*switch light on*)
IF i_bSwitchOn OR (io_TypeLED.fpSwitchOnOff.Q AND NOT io_TypeLED.bLight) THEN
	io_TypeLED.Switch_ON := TRUE;
END_IF

(*switch light off*)
IF i_bSwitchOff OR (io_TypeLED.fpSwitchOnOff.Q AND io_TypeLED.bLight) THEN
	io_TypeLED.Switch_ON := FALSE;
END_IF

io_TypeLED.fbDimmer2Switch(
	bSwitchDimmUp:= FALSE,
	bSwitchDimmDown:= FALSE,
	bOn:= io_TypeLED.Switch_ON,
	bOff:= NOT io_TypeLED.Switch_ON,
	bSetDimmValue:= FALSE,
	nDimmValue:= 0,
	tSwitchOverTime:=T#300MS ,
	tDimmTime:= REAL_TO_TIME(io_TypeLED.Config.tDimmTime),
	bMemoryModeOn:= TRUE,
	nOnValueWithoutMemoryMode:= 0,
	bDimmOnMode:= io_TypeLED.Config.bDimmOnMode,
	tDimmOnTime:= REAL_TO_TIME(io_TypeLED.Config.tDimmOnTime),
	bDimmOffMode:= io_TypeLED.Config.bDimmOffMode,
	tDimmOffTime:= REAL_TO_TIME(io_TypeLED.Config.tDimmOffTime),
	nOutMin:= 0,
	nOutMax:=100,
	bLight=> io_TypeLED.bLight);

io_TypeLED.Brightness := REAL_TO_BYTE(UINT_TO_REAL(io_TypeLED.fbDimmer2Switch.nOut)/100*io_TypeLED.Config.Brightness_MAX*(io_TypeLED.Value/100));
END_PROGRAM

(* POU Imported fileses from libraries/DEC1, ST *)
FUNCTION DEC1 : INT
VAR_INPUT
	X : INT;
	N : INT;
END_VAR


(*
version 1.1	27. oct. 2008
programmer 	hugo
tested by	oscat

This is a decrement function which decrements the variable X by 1 and if 0 is reached, it begins with N-1 again.
_dec1(X,3) will generate 2,1,0,2,...

*)
IF X = 0 THEN
	DEC1 := N - 1;
ELSE
	DEC1 := X - 1;
END_IF;


(* this is a very elegant version but 50% slower
X := (X - 1 + N) MOD N;
*)


(* revision history
hm	13. oct. 2008	rev 1.0
	original version

hm	27. oct. 2008	rev 1.1
	added statement to return value for compatibility reasons

*)
END_FUNCTION

(* POU Imported fileses from libraries/INC1, ST *)
FUNCTION INC1 : INT
VAR_INPUT
	X : INT;
	N : INT;
END_VAR



(*
version 1.2	23. feb. 2009
programmer 	hugo
tested by	oscat

This is a increment function which increments the variable X by 1 and if N is reached, it begins with 0 instead of N again.
inc1(X,3) will generate 0,1,2,0,1,.....

*)
IF X >= N - 1 THEN
	INC1 := 0;
ELSE
	INC1 := X + 1;
END_IF;



(* revision history
hm	13. oct. 2008	rev 1.0
	original version

hm	22. oct. 2008	rev 1.1
	added statement to return value for compatibility reasons

hm	23. feb. 2009	rev 1.2
 	when inc1 is called with X >= N inc will continue with 0
*)
END_FUNCTION

(* POU Own PRG's and FB's/PRG_FIFO_10080, ST *)
FUNCTION_BLOCK PRG_FIFO_10080
VAR_INPUT
	REALin : REAL;
	tTime:TIMESTRUCT;
	E : BOOL := TRUE;
	RD : BOOL;
	WD : BOOL;
	RST : BOOL;
END_VAR
VAR_OUTPUT
	REALout : REAL;
	YEARout : WORD;
	MONTHout : WORD;
	DAYout : WORD;
	HOURout : WORD;
	MINUTEout : WORD;
	EMPTY : BOOL := TRUE;
	FULL : BOOL;
END_VAR
VAR
	fifo : ARRAY[0..n] OF REAL;
	fifoYEAR : ARRAY[0..n] OF WORD;
	fifoMONTH : ARRAY[0..n] OF WORD;
	fifoDAY : ARRAY[0..n] OF WORD;
	fifoHOUR : ARRAY[0..n] OF WORD;
	fifoMINUTE : ARRAY[0..n] OF WORD;
	fifoSECOND : ARRAY[0..n] OF WORD;
	p : INT;
END_VAR
VAR CONSTANT
	n : INT := 10080;	(* changing this value will chage the number of stored elements in the fifo *)
END_VAR

(*
version 2.0	24. jul. 2009
programmer 	hugo
tested by		oscat

32 Dword FIFO memory
*)
IF RST THEN
	p := 0;
	FULL := FALSE;
	EMPTY := TRUE;
	REALout := 0;
	YEARout :=0;
	MONTHout :=0;
	DAYout := 0;
	HOURout := 0;
	MINUTEout := 0;
ELSIF E THEN
	IF NOT EMPTY AND RD THEN
		fifo[p] := 0;
		fifoYEAR[p] := 0;
		fifoMONTH[p] := 0;
		fifoDAY[p] := 0;
		fifoHOUR[p] := 0;
		fifoMINUTE[p] := 0;
		p := DEC1(p,n);
		REALout := fifo[p];
		YEARout := fifoYEAR[p];
		MONTHout := fifoMONTH[p];
		DAYout := fifoDAY[p];
		HOURout := fifoHOUR[p];
		MINUTEout := fifoMINUTE[p];
		EMPTY := p = 0;
		FULL := FALSE;
	END_IF;
	IF NOT FULL AND WD THEN
		fifo[p] := REALin;
		fifoYEAR[p] := tTime.wYear;
		fifoMONTH[p] := tTime.wMonth;
		fifoDAY[p] := tTime.wDay;
		fifoHOUR[p] := tTime.wHour;
		fifoMINUTE[p] := tTime.wMinute;
		REALout := fifo[p];
		YEARout := fifoYEAR[p];
		MONTHout := fifoMONTH[p];
		DAYout := fifoDAY[p];
		HOURout := fifoHOUR[p];
		MINUTEout := fifoMINUTE[p];
		p := INC1(p,n);
		FULL := p = n;
		EMPTY := FALSE;
	END_IF;
END_IF;




(* revision history
hm	4. aug. 2006	rev 1.0
	original version

hm	19. feb 2008	rev 1.1
	performance improvements

hm	17. oct. 2008	rev 1.2
	improved performance

ks	27. oct. 2008 rev 1.3
	improved code

hm	14. mar. 2009	rev 1.4
	removed double assignments

hm 24. jul. 2009	rev 2.0
	chaged inputs E and WR to E, WD and WR
	allow read and write in one cycle

*)
END_FUNCTION_BLOCK
